(* Logix 5000 project; controller reports 1756-L63 rev 20.15; software revision 20.04; part 46 of 52 *)

        [142].log_data[50].min := 2.0290048, [142].log_data[50].max := 2.1358266, [142].log_data[50].total := 7520.501, [142].log_data[50].time := 3600.0, [142].log_data[50].minminute := 14, [142].log_data[50].maxminute := 21, [142].log_data[50].valid := 1, [142].log_data[51].time := 3600.0, [142].log_data[51].valid := 1, [142].log_data[52].min := -2.9000015, [142].log_data[52].max := 0.11999512, [142].log_data[52].total := -7928.3423, [142].log_data[52].time := 3600.0, [142].log_data[52].minminute := 8, [142].log_data[52].maxminute := 7, [142].log_data[52].valid := 1, [142].log_data[53].min := -2.4600067, [142].log_data[53].max := 0.38000488, [142].log_data[53].total := -6926.5454, [142].log_data[53].time := 3600.0, [142].log_data[53].minminute := 24, [142].log_data[53].maxminute := 13, [142].log_data[53].valid := 1, [142].log_data[54].max := 0.524, [142].log_data[54].total := 1245.6982, [142].log_data[54].time := 3600.0, [142].log_data[54].minminute := 7, [142].log_data[54].maxminute := 8, [142].log_data[54].valid := 1, [142].log_data[55].max := 0.5415, [142].log_data[55].total := 1217.0897, [142].log_data[55].time := 3600.0, [142].log_data[55].minminute := 2, [142].log_data[55].maxminute := 24, [142].log_data[55].valid := 1, [142].log_data[56].min := 0.15906787, [142].log_data[56].max := 0.15965673, [142].log_data[56].total := 573.5303, [142].log_data[56].time := 3600.0, [142].log_data[56].minminute := 45, [142].log_data[56].maxminute := 33, [142].log_data[56].valid := 1, [142].log_data[57].min := 0.19345811, [142].log_data[57].max := 0.19534253, [142].log_data[57].total := 701.22565, [142].log_data[57].time := 3600.0, [142].log_data[57].minminute := 53, [142].log_data[57].valid := 1, [142].log_data[58].time := 3600.0, [142].log_data[58].valid := 1, [142].log_data[59].time := 3600.0, [142].log_data[59].valid := 1, [142].log_data[60].valid := 1, [142].log_data[61].valid := 1, [142].log_data[62].valid := 1, [142].log_data[63].valid := 1, [142].log_data[64].valid := 1, [142].log_data[65].valid := 1, [142].log_data[66].valid := 1, [142].log_data[67].valid := 1,
        [142].log_data[68].valid := 1, [142].log_data[69].valid := 1, [142].log_data[70].valid := 1, [142].log_data[71].valid := 1, [142].log_data[72].valid := 1, [142].log_data[73].valid := 1, [142].log_data[74].valid := 1, [142].log_data[75].valid := 1, [142].log_data[76].valid := 1, [142].log_data[77].valid := 1, [142].log_data[78].valid := 1, [142].log_data[79].valid := 1, [142].log_data[80].valid := 1, [142].log_data[81].valid := 1, [142].log_data[82].valid := 1, [142].log_data[83].valid := 1, [142].log_data[84].valid := 1, [142].log_data[85].valid := 1, [142].log_data[86].valid := 1, [142].log_data[87].valid := 1, [142].log_data[88].valid := 1, [142].log_data[89].valid := 1, [142].log_data[90].valid := 1, [142].log_data[91].valid := 1, [142].log_data[92].valid := 1, [142].log_data[93].valid := 1, [142].log_data[94].valid := 1, [142].log_data[95].valid := 1, [142].log_data[96].valid := 1, [142].log_data[97].valid := 1, [142].log_data[98].valid := 1, [142].log_data[99].valid := 1, [142].log_data[100].valid := 1, [142].log_data[101].valid := 1, [142].log_data[102].valid := 1, [142].log_data[103].valid := 1, [142].log_data[104].valid := 1, [142].log_data[105].valid := 1, [142].log_data[106].valid := 1, [142].log_data[107].valid := 1, [142].log_data[108].valid := 1, [142].log_data[109].valid := 1, [142].log_data[110].valid := 1, [142].log_data[111].valid := 1, [142].log_data[112].valid := 1, [142].log_data[113].valid := 1, [142].log_data[114].valid := 1, [142].log_data[115].valid := 1, [142].log_data[116].valid := 1, [142].log_data[117].valid := 1, [142].log_data[118].valid := 1, [142].log_data[119].valid := 1, [142].log_data[120].valid := 1, [142].log_data[121].valid := 1, [142].log_data[122].valid := 1, [142].log_data[123].valid := 1, [142].log_data[124].valid := 1, [142].time.Year := 2023, [142].time.Month := 1, [142].time.Day := 19,
        [142].time.Hour := 1, [142].time.Minute := 59, [142].time.Second := 59, [143].log_data[0].min := 1.0, [143].log_data[0].max := 1.0, [143].log_data[0].total := 3600.0, [143].log_data[0].time := 3600.0, [143].log_data[0].valid := 1, [143].log_data[1].time := 3600.0, [143].log_data[1].valid := 1, [143].log_data[2].time := 3600.0, [143].log_data[2].valid := 1, [143].log_data[3].time := 3600.0, [143].log_data[3].valid := 1, [143].log_data[4].time := 3600.0, [143].log_data[4].valid := 1, [143].log_data[5].time := 3600.0, [143].log_data[5].valid := 1, [143].log_data[6].time := 3600.0, [143].log_data[6].valid := 1, [143].log_data[7].time := 3600.0, [143].log_data[7].valid := 1, [143].log_data[8].min := 1.0, [143].log_data[8].max := 1.0, [143].log_data[8].total := 3600.0, [143].log_data[8].time := 3600.0, [143].log_data[8].valid := 1, [143].log_data[9].min := 1.0, [143].log_data[9].max := 1.0, [143].log_data[9].total := 3600.0, [143].log_data[9].time := 3600.0, [143].log_data[9].valid := 1, [143].log_data[10].min := 1.0, [143].log_data[10].max := 1.0, [143].log_data[10].total := 3600.0, [143].log_data[10].time := 3600.0, [143].log_data[10].valid := 1, [143].log_data[11].time := 3600.0, [143].log_data[11].valid := 1, [143].log_data[12].min := 1.0, [143].log_data[12].max := 1.0, [143].log_data[12].total := 3600.0, [143].log_data[12].time := 3600.0, [143].log_data[12].valid := 1, [143].log_data[13].min := 1.0, [143].log_data[13].max := 1.0, [143].log_data[13].total := 3600.0, [143].log_data[13].time := 3600.0, [143].log_data[13].valid := 1, [143].log_data[14].time := 3600.0, [143].log_data[14].valid := 1, [143].log_data[15].time := 3600.0, [143].log_data[15].valid := 1, [143].log_data[16].time := 3600.0, [143].log_data[16].valid := 1, [143].log_data[17].min := 1.0, [143].log_data[17].max := 1.0, [143].log_data[17].total := 3600.0, [143].log_data[17].time := 3600.0, [143].log_data[17].valid := 1,
        [143].log_data[18].time := 3600.0, [143].log_data[18].valid := 1, [143].log_data[19].time := 3600.0, [143].log_data[19].valid := 1, [143].log_data[20].time := 3600.0, [143].log_data[20].valid := 1, [143].log_data[21].min := 1.0, [143].log_data[21].max := 1.0, [143].log_data[21].total := 3600.0, [143].log_data[21].time := 3600.0, [143].log_data[21].valid := 1, [143].log_data[22].time := 3600.0, [143].log_data[22].valid := 1, [143].log_data[23].time := 3600.0, [143].log_data[23].valid := 1, [143].log_data[24].time := 3600.0, [143].log_data[24].valid := 1, [143].log_data[25].time := 3600.0, [143].log_data[25].valid := 1, [143].log_data[26].time := 3600.0, [143].log_data[26].valid := 1, [143].log_data[27].time := 3600.0, [143].log_data[27].valid := 1, [143].log_data[28].time := 3600.0, [143].log_data[28].valid := 1, [143].log_data[29].min := 1.0, [143].log_data[29].max := 1.0, [143].log_data[29].total := 3600.0, [143].log_data[29].time := 3600.0, [143].log_data[29].valid := 1, [143].log_data[30].min := 1.0, [143].log_data[30].max := 1.0, [143].log_data[30].total := 3600.0, [143].log_data[30].time := 3600.0, [143].log_data[30].valid := 1, [143].log_data[31].max := 1.0, [143].log_data[31].total := 1464.2471, [143].log_data[31].time := 3600.0, [143].log_data[31].maxminute := 11, [143].log_data[31].valid := 1, [143].log_data[32].max := 1.0, [143].log_data[32].total := 1629.998, [143].log_data[32].time := 3600.0, [143].log_data[32].maxminute := 1, [143].log_data[32].valid := 1, [143].log_data[33].time := 3600.0, [143].log_data[33].valid := 1, [143].log_data[34].time := 3600.0, [143].log_data[34].valid := 1, [143].log_data[35].max := 1.0, [143].log_data[35].total := 1629.498, [143].log_data[35].time := 3600.0, [143].log_data[35].maxminute := 6, [143].log_data[35].valid := 1, [143].log_data[36].max := 1.0, [143].log_data[36].total := 1440.7471, [143].log_data[36].time := 3600.0, [143].log_data[36].minminute := 5, [143].log_data[36].valid := 1, [143].log_data[37].time := 3600.0,
        [143].log_data[37].valid := 1, [143].log_data[38].time := 3600.0, [143].log_data[38].valid := 1, [143].log_data[39].min := 0.9961195, [143].log_data[39].max := 1.0054238, [143].log_data[39].total := 3604.2942, [143].log_data[39].time := 3600.0, [143].log_data[39].minminute := 29, [143].log_data[39].maxminute := 50, [143].log_data[39].valid := 1, [143].log_data[40].min := 7.602789, [143].log_data[40].max := 7.622027, [143].log_data[40].total := 27405.582, [143].log_data[40].time := 3600.0, [143].log_data[40].minminute := 5, [143].log_data[40].maxminute := 10, [143].log_data[40].valid := 1, [143].log_data[41].min := 0.02273633, [143].log_data[41].max := 0.023128908, [143].log_data[41].total := 82.62436, [143].log_data[41].time := 3600.0, [143].log_data[41].valid := 1, [143].log_data[42].min := 2.291525, [143].log_data[42].max := 2.296236, [143].log_data[42].total := 8257.919, [143].log_data[42].time := 3600.0, [143].log_data[42].minminute := 2, [143].log_data[42].maxminute := 20, [143].log_data[42].valid := 1, [143].log_data[43].min := -0.27999878, [143].log_data[43].max := -0.26000214, [143].log_data[43].total := -1007.4526, [143].log_data[43].time := 3600.0, [143].log_data[43].maxminute := 8, [143].log_data[43].valid := 1, [143].log_data[44].min := -0.3199997, [143].log_data[44].max := -0.30000305, [143].log_data[44].total := -1092.692, [143].log_data[44].time := 3600.0, [143].log_data[44].valid := 1, [143].log_data[45].time := 3600.0, [143].log_data[45].valid := 1, [143].log_data[46].time := 3600.0, [143].log_data[46].valid := 1, [143].log_data[47].time := 3600.0, [143].log_data[47].valid := 1, [143].log_data[48].min := 6.7536335, [143].log_data[48].max := 6.7967777, [143].log_data[48].total := 24351.693, [143].log_data[48].time := 3600.0, [143].log_data[48].minminute := 54, [143].log_data[48].maxminute := 1, [143].log_data[48].valid := 1, [143].log_data[49].min := 8.710789, [143].log_data[49].max := 9.616479, [143].log_data[49].total := 33962.16, [143].log_data[49].time := 3600.0, [143].log_data[49].maxminute := 42, [143].log_data[49].valid := 1, [143].log_data[50].min := 2.0009744,
        [143].log_data[50].max := 2.0865965, [143].log_data[50].total := 7354.9937, [143].log_data[50].time := 3600.0, [143].log_data[50].minminute := 59, [143].log_data[50].valid := 1, [143].log_data[51].time := 3600.0, [143].log_data[51].valid := 1, [143].log_data[52].min := -2.8199997, [143].log_data[52].max := 0.11999512, [143].log_data[52].total := -7782.8364, [143].log_data[52].time := 3600.0, [143].log_data[52].minminute := 32, [143].log_data[52].maxminute := 11, [143].log_data[52].valid := 1, [143].log_data[53].min := -2.6200027, [143].log_data[53].max := 0.33999634, [143].log_data[53].total := -6983.5625, [143].log_data[53].time := 3600.0, [143].log_data[53].minminute := 48, [143].log_data[53].maxminute := 16, [143].log_data[53].valid := 1, [143].log_data[54].max := 0.5265, [143].log_data[54].total := 1226.1595, [143].log_data[54].time := 3600.0, [143].log_data[54].maxminute := 32, [143].log_data[54].valid := 1, [143].log_data[55].max := 0.55149996, [143].log_data[55].total := 1217.2601, [143].log_data[55].time := 3600.0, [143].log_data[55].minminute := 5, [143].log_data[55].maxminute := 48, [143].log_data[55].valid := 1, [143].log_data[56].min := 0.15918565, [143].log_data[56].max := 0.15961748, [143].log_data[56].total := 573.6516, [143].log_data[56].time := 3600.0, [143].log_data[56].maxminute := 29, [143].log_data[56].valid := 1, [143].log_data[57].min := 0.1933796, [143].log_data[57].max := 0.19381143, [143].log_data[57].total := 696.8782, [143].log_data[57].time := 3600.0, [143].log_data[57].minminute := 28, [143].log_data[57].maxminute := 7, [143].log_data[57].valid := 1, [143].log_data[58].time := 3600.0, [143].log_data[58].valid := 1, [143].log_data[59].time := 3600.0, [143].log_data[59].valid := 1, [143].log_data[60].valid := 1, [143].log_data[61].valid := 1, [143].log_data[62].valid := 1, [143].log_data[63].valid := 1, [143].log_data[64].valid := 1, [143].log_data[65].valid := 1, [143].log_data[66].valid := 1, [143].log_data[67].valid := 1, [143].log_data[68].valid := 1, [143].log_data[69].valid := 1, [143].log_data[70].valid := 1,
        [143].log_data[71].valid := 1, [143].log_data[72].valid := 1, [143].log_data[73].valid := 1, [143].log_data[74].valid := 1, [143].log_data[75].valid := 1, [143].log_data[76].valid := 1, [143].log_data[77].valid := 1, [143].log_data[78].valid := 1, [143].log_data[79].valid := 1, [143].log_data[80].valid := 1, [143].log_data[81].valid := 1, [143].log_data[82].valid := 1, [143].log_data[83].valid := 1, [143].log_data[84].valid := 1, [143].log_data[85].valid := 1, [143].log_data[86].valid := 1, [143].log_data[87].valid := 1, [143].log_data[88].valid := 1, [143].log_data[89].valid := 1, [143].log_data[90].valid := 1, [143].log_data[91].valid := 1, [143].log_data[92].valid := 1, [143].log_data[93].valid := 1, [143].log_data[94].valid := 1, [143].log_data[95].valid := 1, [143].log_data[96].valid := 1, [143].log_data[97].valid := 1, [143].log_data[98].valid := 1, [143].log_data[99].valid := 1, [143].log_data[100].valid := 1, [143].log_data[101].valid := 1, [143].log_data[102].valid := 1, [143].log_data[103].valid := 1, [143].log_data[104].valid := 1, [143].log_data[105].valid := 1, [143].log_data[106].valid := 1, [143].log_data[107].valid := 1, [143].log_data[108].valid := 1, [143].log_data[109].valid := 1, [143].log_data[110].valid := 1, [143].log_data[111].valid := 1, [143].log_data[112].valid := 1, [143].log_data[113].valid := 1, [143].log_data[114].valid := 1, [143].log_data[115].valid := 1, [143].log_data[116].valid := 1, [143].log_data[117].valid := 1, [143].log_data[118].valid := 1, [143].log_data[119].valid := 1, [143].log_data[120].valid := 1, [143].log_data[121].valid := 1, [143].log_data[122].valid := 1, [143].log_data[123].valid := 1, [143].log_data[124].valid := 1, [143].time.Year := 2023, [143].time.Month := 1, [143].time.Day := 19, [143].time.Hour := 2, [143].time.Minute := 59, [143].time.Second := 59,
        [144].log_data[0].min := 1.0, [144].log_data[0].max := 1.0, [144].log_data[0].total := 3600.0, [144].log_data[0].time := 3600.0, [144].log_data[0].valid := 1, [144].log_data[1].time := 3600.0, [144].log_data[1].valid := 1, [144].log_data[2].time := 3600.0, [144].log_data[2].valid := 1, [144].log_data[3].time := 3600.0, [144].log_data[3].valid := 1, [144].log_data[4].time := 3600.0, [144].log_data[4].valid := 1, [144].log_data[5].time := 3600.0, [144].log_data[5].valid := 1, [144].log_data[6].time := 3600.0, [144].log_data[6].valid := 1, [144].log_data[7].time := 3600.0, [144].log_data[7].valid := 1, [144].log_data[8].max := 1.0, [144].log_data[8].total := 22.251, [144].log_data[8].time := 3600.0, [144].log_data[8].valid := 1, [144].log_data[9].max := 1.0, [144].log_data[9].total := 22.251, [144].log_data[9].time := 3600.0, [144].log_data[9].valid := 1, [144].log_data[10].min := 1.0, [144].log_data[10].max := 1.0, [144].log_data[10].total := 3600.0, [144].log_data[10].time := 3600.0, [144].log_data[10].valid := 1, [144].log_data[11].time := 3600.0, [144].log_data[11].valid := 1, [144].log_data[12].min := 1.0, [144].log_data[12].max := 1.0, [144].log_data[12].total := 3600.0, [144].log_data[12].time := 3600.0, [144].log_data[12].valid := 1, [144].log_data[13].min := 1.0, [144].log_data[13].max := 1.0, [144].log_data[13].total := 3600.0, [144].log_data[13].time := 3600.0, [144].log_data[13].valid := 1, [144].log_data[14].time := 3600.0, [144].log_data[14].valid := 1, [144].log_data[15].time := 3600.0, [144].log_data[15].valid := 1, [144].log_data[16].time := 3600.0, [144].log_data[16].valid := 1, [144].log_data[17].min := 1.0, [144].log_data[17].max := 1.0, [144].log_data[17].total := 3600.0, [144].log_data[17].time := 3600.0, [144].log_data[17].valid := 1, [144].log_data[18].time := 3600.0, [144].log_data[18].valid := 1, [144].log_data[19].time := 3600.0, [144].log_data[19].valid := 1, [144].log_data[20].time := 3600.0,
        [144].log_data[20].valid := 1, [144].log_data[21].min := 1.0, [144].log_data[21].max := 1.0, [144].log_data[21].total := 3600.0, [144].log_data[21].time := 3600.0, [144].log_data[21].valid := 1, [144].log_data[22].time := 3600.0, [144].log_data[22].valid := 1, [144].log_data[23].time := 3600.0, [144].log_data[23].valid := 1, [144].log_data[24].time := 3600.0, [144].log_data[24].valid := 1, [144].log_data[25].time := 3600.0, [144].log_data[25].valid := 1, [144].log_data[26].time := 3600.0, [144].log_data[26].valid := 1, [144].log_data[27].time := 3600.0, [144].log_data[27].valid := 1, [144].log_data[28].time := 3600.0, [144].log_data[28].valid := 1, [144].log_data[29].min := 1.0, [144].log_data[29].max := 1.0, [144].log_data[29].total := 3600.0, [144].log_data[29].time := 3600.0, [144].log_data[29].valid := 1, [144].log_data[30].min := 1.0, [144].log_data[30].max := 1.0, [144].log_data[30].total := 3600.0, [144].log_data[30].time := 3600.0, [144].log_data[30].valid := 1, [144].log_data[31].max := 1.0, [144].log_data[31].total := 26.0, [144].log_data[31].time := 3600.0, [144].log_data[31].valid := 1, [144].log_data[32].time := 3600.0, [144].log_data[32].valid := 1, [144].log_data[33].time := 3600.0, [144].log_data[33].valid := 1, [144].log_data[34].time := 3600.0, [144].log_data[34].valid := 1, [144].log_data[35].time := 3600.0, [144].log_data[35].valid := 1, [144].log_data[36].max := 1.0, [144].log_data[36].total := 26.0, [144].log_data[36].time := 3600.0, [144].log_data[36].valid := 1, [144].log_data[37].time := 3600.0, [144].log_data[37].valid := 1, [144].log_data[38].time := 3600.0, [144].log_data[38].valid := 1, [144].log_data[39].min := 0.99623734, [144].log_data[39].max := 1.0056593, [144].log_data[39].total := 3605.3367, [144].log_data[39].time := 3600.0, [144].log_data[39].minminute := 48, [144].log_data[39].maxminute := 56, [144].log_data[39].valid := 1, [144].log_data[40].min := 7.5972934, [144].log_data[40].max := 7.6363163, [144].log_data[40].total := 27399.168,
        [144].log_data[40].time := 3600.0, [144].log_data[40].minminute := 26, [144].log_data[40].maxminute := 33, [144].log_data[40].valid := 1, [144].log_data[41].min := 0.02273633, [144].log_data[41].max := 0.023128908, [144].log_data[41].total := 82.62523, [144].log_data[41].time := 3600.0, [144].log_data[41].valid := 1, [144].log_data[42].min := 2.2910538, [144].log_data[42].max := 2.2958827, [144].log_data[42].total := 8257.894, [144].log_data[42].time := 3600.0, [144].log_data[42].minminute := 22, [144].log_data[42].maxminute := 8, [144].log_data[42].valid := 1, [144].log_data[43].min := -0.27999878, [144].log_data[43].max := -0.26000214, [144].log_data[43].total := -1007.2367, [144].log_data[43].time := 3600.0, [144].log_data[43].valid := 1, [144].log_data[44].min := -0.3199997, [144].log_data[44].max := -0.30000305, [144].log_data[44].total := -1086.3679, [144].log_data[44].time := 3600.0, [144].log_data[44].valid := 1, [144].log_data[45].time := 3600.0, [144].log_data[45].valid := 1, [144].log_data[46].time := 3600.0, [144].log_data[46].valid := 1, [144].log_data[47].time := 3600.0, [144].log_data[47].valid := 1, [144].log_data[48].min := 6.7519846, [144].log_data[48].max := 6.768473, [144].log_data[48].total := 24336.852, [144].log_data[48].time := 3600.0, [144].log_data[48].minminute := 2, [144].log_data[48].maxminute := 55, [144].log_data[48].valid := 1, [144].log_data[49].min := 9.541692, [144].log_data[49].max := 9.602148, [144].log_data[49].total := 34445.23, [144].log_data[49].time := 3600.0, [144].log_data[49].minminute := 5, [144].log_data[49].maxminute := 7, [144].log_data[49].valid := 1, [144].log_data[50].min := 1.9997966, [144].log_data[50].max := 2.110623, [144].log_data[50].total := 7565.291, [144].log_data[50].time := 3600.0, [144].log_data[50].maxminute := 56, [144].log_data[50].valid := 1, [144].log_data[51].time := 3600.0, [144].log_data[51].valid := 1, [144].log_data[52].min := -2.6399994, [144].log_data[52].max := -0.08000183, [144].log_data[52].total := -5223.154, [144].log_data[52].time := 3600.0, [144].log_data[52].valid := 1, [144].log_data[53].min := -2.4200058,
        [144].log_data[53].max := -0.16000366, [144].log_data[53].total := -4604.705, [144].log_data[53].time := 3600.0, [144].log_data[53].valid := 1, [144].log_data[54].max := 0.43400002, [144].log_data[54].total := 10.802108, [144].log_data[54].time := 3600.0, [144].log_data[54].valid := 1, [144].log_data[55].max := 0.4145, [144].log_data[55].total := 10.702488, [144].log_data[55].time := 3600.0, [144].log_data[55].valid := 1, [144].log_data[56].min := 0.15918565, [144].log_data[56].max := 0.15961748, [144].log_data[56].total := 573.69305, [144].log_data[56].time := 3600.0, [144].log_data[56].minminute := 11, [144].log_data[56].maxminute := 36, [144].log_data[56].valid := 1, [144].log_data[57].min := 0.19334033, [144].log_data[57].max := 0.19377217, [144].log_data[57].total := 696.698, [144].log_data[57].time := 3600.0, [144].log_data[57].minminute := 2, [144].log_data[57].maxminute := 16, [144].log_data[57].valid := 1, [144].log_data[58].time := 3600.0, [144].log_data[58].valid := 1, [144].log_data[59].time := 3600.0, [144].log_data[59].valid := 1, [144].log_data[60].valid := 1, [144].log_data[61].valid := 1, [144].log_data[62].valid := 1, [144].log_data[63].valid := 1, [144].log_data[64].valid := 1, [144].log_data[65].valid := 1, [144].log_data[66].valid := 1, [144].log_data[67].valid := 1, [144].log_data[68].valid := 1, [144].log_data[69].valid := 1, [144].log_data[70].valid := 1, [144].log_data[71].valid := 1, [144].log_data[72].valid := 1, [144].log_data[73].valid := 1, [144].log_data[74].valid := 1, [144].log_data[75].valid := 1, [144].log_data[76].valid := 1, [144].log_data[77].valid := 1, [144].log_data[78].valid := 1, [144].log_data[79].valid := 1, [144].log_data[80].valid := 1, [144].log_data[81].valid := 1, [144].log_data[82].valid := 1, [144].log_data[83].valid := 1, [144].log_data[84].valid := 1, [144].log_data[85].valid := 1, [144].log_data[86].valid := 1, [144].log_data[87].valid := 1, [144].log_data[88].valid := 1, [144].log_data[89].valid := 1,
        [144].log_data[90].valid := 1, [144].log_data[91].valid := 1, [144].log_data[92].valid := 1, [144].log_data[93].valid := 1, [144].log_data[94].valid := 1, [144].log_data[95].valid := 1, [144].log_data[96].valid := 1, [144].log_data[97].valid := 1, [144].log_data[98].valid := 1, [144].log_data[99].valid := 1, [144].log_data[100].valid := 1, [144].log_data[101].valid := 1, [144].log_data[102].valid := 1, [144].log_data[103].valid := 1, [144].log_data[104].valid := 1, [144].log_data[105].valid := 1, [144].log_data[106].valid := 1, [144].log_data[107].valid := 1, [144].log_data[108].valid := 1, [144].log_data[109].valid := 1, [144].log_data[110].valid := 1, [144].log_data[111].valid := 1, [144].log_data[112].valid := 1, [144].log_data[113].valid := 1, [144].log_data[114].valid := 1, [144].log_data[115].valid := 1, [144].log_data[116].valid := 1, [144].log_data[117].valid := 1, [144].log_data[118].valid := 1, [144].log_data[119].valid := 1, [144].log_data[120].valid := 1, [144].log_data[121].valid := 1, [144].log_data[122].valid := 1, [144].log_data[123].valid := 1, [144].log_data[124].valid := 1, [144].time.Year := 2023, [144].time.Month := 1, [144].time.Day := 19, [144].time.Hour := 3, [144].time.Minute := 59, [144].time.Second := 59, [145].log_data[0].min := 1.0, [145].log_data[0].max := 1.0, [145].log_data[0].total := 3600.0, [145].log_data[0].time := 3600.0, [145].log_data[0].valid := 1, [145].log_data[1].time := 3600.0, [145].log_data[1].valid := 1, [145].log_data[2].time := 3600.0, [145].log_data[2].valid := 1, [145].log_data[3].time := 3600.0, [145].log_data[3].valid := 1, [145].log_data[4].time := 3600.0, [145].log_data[4].valid := 1, [145].log_data[5].time := 3600.0, [145].log_data[5].valid := 1, [145].log_data[6].time := 3600.0, [145].log_data[6].valid := 1, [145].log_data[7].time := 3600.0, [145].log_data[7].valid := 1,
        [145].log_data[8].time := 3600.0, [145].log_data[8].valid := 1, [145].log_data[9].time := 3600.0, [145].log_data[9].valid := 1, [145].log_data[10].min := 1.0, [145].log_data[10].max := 1.0, [145].log_data[10].total := 3600.0, [145].log_data[10].time := 3600.0, [145].log_data[10].valid := 1, [145].log_data[11].time := 3600.0, [145].log_data[11].valid := 1, [145].log_data[12].min := 1.0, [145].log_data[12].max := 1.0, [145].log_data[12].total := 3600.0, [145].log_data[12].time := 3600.0, [145].log_data[12].valid := 1, [145].log_data[13].min := 1.0, [145].log_data[13].max := 1.0, [145].log_data[13].total := 3600.0, [145].log_data[13].time := 3600.0, [145].log_data[13].valid := 1, [145].log_data[14].time := 3600.0, [145].log_data[14].valid := 1, [145].log_data[15].time := 3600.0, [145].log_data[15].valid := 1, [145].log_data[16].time := 3600.0, [145].log_data[16].valid := 1, [145].log_data[17].min := 1.0, [145].log_data[17].max := 1.0, [145].log_data[17].total := 3600.0, [145].log_data[17].time := 3600.0, [145].log_data[17].valid := 1, [145].log_data[18].time := 3600.0, [145].log_data[18].valid := 1, [145].log_data[19].time := 3600.0, [145].log_data[19].valid := 1, [145].log_data[20].time := 3600.0, [145].log_data[20].valid := 1, [145].log_data[21].min := 1.0, [145].log_data[21].max := 1.0, [145].log_data[21].total := 3600.0, [145].log_data[21].time := 3600.0, [145].log_data[21].valid := 1, [145].log_data[22].time := 3600.0, [145].log_data[22].valid := 1, [145].log_data[23].time := 3600.0, [145].log_data[23].valid := 1, [145].log_data[24].time := 3600.0, [145].log_data[24].valid := 1, [145].log_data[25].time := 3600.0, [145].log_data[25].valid := 1, [145].log_data[26].time := 3600.0, [145].log_data[26].valid := 1, [145].log_data[27].time := 3600.0, [145].log_data[27].valid := 1, [145].log_data[28].time := 3600.0, [145].log_data[28].valid := 1, [145].log_data[29].min := 1.0, [145].log_data[29].max := 1.0, [145].log_data[29].total := 3600.0,
        [145].log_data[29].time := 3600.0, [145].log_data[29].valid := 1, [145].log_data[30].min := 1.0, [145].log_data[30].max := 1.0, [145].log_data[30].total := 3600.0, [145].log_data[30].time := 3600.0, [145].log_data[30].valid := 1, [145].log_data[31].time := 3600.0, [145].log_data[31].valid := 1, [145].log_data[32].time := 3600.0, [145].log_data[32].valid := 1, [145].log_data[33].time := 3600.0, [145].log_data[33].valid := 1, [145].log_data[34].time := 3600.0, [145].log_data[34].valid := 1, [145].log_data[35].time := 3600.0, [145].log_data[35].valid := 1, [145].log_data[36].time := 3600.0, [145].log_data[36].valid := 1, [145].log_data[37].time := 3600.0, [145].log_data[37].valid := 1, [145].log_data[38].time := 3600.0, [145].log_data[38].valid := 1, [145].log_data[39].min := 0.9967084, [145].log_data[39].max := 1.0062482, [145].log_data[39].total := 3605.411, [145].log_data[39].time := 3600.0, [145].log_data[39].maxminute := 1, [145].log_data[39].valid := 1, [145].log_data[40].min := 7.6030645, [145].log_data[40].max := 7.6250496, [145].log_data[40].total := 27410.46, [145].log_data[40].time := 3600.0, [145].log_data[40].minminute := 2, [145].log_data[40].maxminute := 3, [145].log_data[40].valid := 1, [145].log_data[41].min := 0.02273633, [145].log_data[41].max := 0.023128908, [145].log_data[41].total := 82.57975, [145].log_data[41].time := 3600.0, [145].log_data[41].valid := 1, [145].log_data[42].min := 2.290936, [145].log_data[42].max := 2.2957647, [145].log_data[42].total := 8257.829, [145].log_data[42].time := 3600.0, [145].log_data[42].minminute := 28, [145].log_data[42].maxminute := 32, [145].log_data[42].valid := 1, [145].log_data[43].min := -0.27999878, [145].log_data[43].max := -0.26000214, [145].log_data[43].total := -1001.4754, [145].log_data[43].time := 3600.0, [145].log_data[43].valid := 1, [145].log_data[44].min := -0.3199997, [145].log_data[44].max := -0.30000305, [145].log_data[44].total := -1080.5452, [145].log_data[44].time := 3600.0, [145].log_data[44].minminute := 6, [145].log_data[44].valid := 1, [145].log_data[45].time := 3600.0,
        [145].log_data[45].valid := 1, [145].log_data[46].time := 3600.0, [145].log_data[46].valid := 1, [145].log_data[47].time := 3600.0, [145].log_data[47].valid := 1, [145].log_data[48].min := 6.7662745, [145].log_data[48].max := 6.778366, [145].log_data[48].total := 24383.604, [145].log_data[48].time := 3600.0, [145].log_data[48].minminute := 1, [145].log_data[48].maxminute := 54, [145].log_data[48].valid := 1, [145].log_data[49].min := 9.56191, [145].log_data[49].max := 9.644745, [145].log_data[49].total := 34582.85, [145].log_data[49].time := 3600.0, [145].log_data[49].minminute := 5, [145].log_data[49].maxminute := 56, [145].log_data[49].valid := 1, [145].log_data[50].min := 2.1029673, [145].log_data[50].max := 2.1119182, [145].log_data[50].total := 7592.0264, [145].log_data[50].time := 3600.0, [145].log_data[50].minminute := 3, [145].log_data[50].maxminute := 54, [145].log_data[50].valid := 1, [145].log_data[51].time := 3600.0, [145].log_data[51].valid := 1, [145].log_data[52].min := -1.7000046, [145].log_data[52].max := -1.4800034, [145].log_data[52].total := -5676.7373, [145].log_data[52].time := 3600.0, [145].log_data[52].minminute := 52, [145].log_data[52].valid := 1, [145].log_data[53].min := -1.3800049, [145].log_data[53].max := -1.2000046, [145].log_data[53].total := -4570.1772, [145].log_data[53].time := 3600.0, [145].log_data[53].minminute := 1, [145].log_data[53].maxminute := 28, [145].log_data[53].valid := 1, [145].log_data[54].time := 3600.0, [145].log_data[54].valid := 1, [145].log_data[55].time := 3600.0, [145].log_data[55].valid := 1, [145].log_data[56].min := 0.15918565, [145].log_data[56].max := 0.15961748, [145].log_data[56].total := 573.68567, [145].log_data[56].time := 3600.0, [145].log_data[56].minminute := 26, [145].log_data[56].maxminute := 14, [145].log_data[56].valid := 1, [145].log_data[57].min := 0.1933796, [145].log_data[57].max := 0.19381143, [145].log_data[57].total := 696.7857, [145].log_data[57].time := 3600.0, [145].log_data[57].minminute := 17, [145].log_data[57].maxminute := 54, [145].log_data[57].valid := 1, [145].log_data[58].time := 3600.0,
        [145].log_data[58].valid := 1, [145].log_data[59].time := 3600.0, [145].log_data[59].valid := 1, [145].log_data[60].valid := 1, [145].log_data[61].valid := 1, [145].log_data[62].valid := 1, [145].log_data[63].valid := 1, [145].log_data[64].valid := 1, [145].log_data[65].valid := 1, [145].log_data[66].valid := 1, [145].log_data[67].valid := 1, [145].log_data[68].valid := 1, [145].log_data[69].valid := 1, [145].log_data[70].valid := 1, [145].log_data[71].valid := 1, [145].log_data[72].valid := 1, [145].log_data[73].valid := 1, [145].log_data[74].valid := 1, [145].log_data[75].valid := 1, [145].log_data[76].valid := 1, [145].log_data[77].valid := 1, [145].log_data[78].valid := 1, [145].log_data[79].valid := 1, [145].log_data[80].valid := 1, [145].log_data[81].valid := 1, [145].log_data[82].valid := 1, [145].log_data[83].valid := 1, [145].log_data[84].valid := 1, [145].log_data[85].valid := 1, [145].log_data[86].valid := 1, [145].log_data[87].valid := 1, [145].log_data[88].valid := 1, [145].log_data[89].valid := 1, [145].log_data[90].valid := 1, [145].log_data[91].valid := 1, [145].log_data[92].valid := 1, [145].log_data[93].valid := 1, [145].log_data[94].valid := 1, [145].log_data[95].valid := 1, [145].log_data[96].valid := 1, [145].log_data[97].valid := 1, [145].log_data[98].valid := 1, [145].log_data[99].valid := 1, [145].log_data[100].valid := 1, [145].log_data[101].valid := 1, [145].log_data[102].valid := 1, [145].log_data[103].valid := 1, [145].log_data[104].valid := 1, [145].log_data[105].valid := 1, [145].log_data[106].valid := 1, [145].log_data[107].valid := 1, [145].log_data[108].valid := 1, [145].log_data[109].valid := 1, [145].log_data[110].valid := 1, [145].log_data[111].valid := 1, [145].log_data[112].valid := 1, [145].log_data[113].valid := 1, [145].log_data[114].valid := 1, [145].log_data[115].valid := 1, [145].log_data[116].valid := 1,
        [145].log_data[117].valid := 1, [145].log_data[118].valid := 1, [145].log_data[119].valid := 1, [145].log_data[120].valid := 1, [145].log_data[121].valid := 1, [145].log_data[122].valid := 1, [145].log_data[123].valid := 1, [145].log_data[124].valid := 1, [145].time.Year := 2023, [145].time.Month := 1, [145].time.Day := 19, [145].time.Hour := 4, [145].time.Minute := 59, [145].time.Second := 59, [146].log_data[0].min := 1.0, [146].log_data[0].max := 1.0, [146].log_data[0].total := 3600.0, [146].log_data[0].time := 3600.0, [146].log_data[0].valid := 1, [146].log_data[1].max := 1.0, [146].log_data[1].total := 527.5, [146].log_data[1].time := 3600.0, [146].log_data[1].maxminute := 34, [146].log_data[1].valid := 1, [146].log_data[2].max := 1.0, [146].log_data[2].total := 524.0, [146].log_data[2].time := 3600.0, [146].log_data[2].maxminute := 34, [146].log_data[2].valid := 1, [146].log_data[3].time := 3600.0, [146].log_data[3].valid := 1, [146].log_data[4].time := 3600.0, [146].log_data[4].valid := 1, [146].log_data[5].max := 1.0, [146].log_data[5].total := 219.0, [146].log_data[5].time := 3600.0, [146].log_data[5].maxminute := 37, [146].log_data[5].valid := 1, [146].log_data[6].time := 3600.0, [146].log_data[6].valid := 1, [146].log_data[7].time := 3600.0, [146].log_data[7].valid := 1, [146].log_data[8].max := 1.0, [146].log_data[8].total := 196.0, [146].log_data[8].time := 3600.0, [146].log_data[8].maxminute := 38, [146].log_data[8].valid := 1, [146].log_data[9].max := 1.0, [146].log_data[9].total := 192.5, [146].log_data[9].time := 3600.0, [146].log_data[9].maxminute := 39, [146].log_data[9].valid := 1, [146].log_data[10].min := 1.0, [146].log_data[10].max := 1.0, [146].log_data[10].total := 3600.0, [146].log_data[10].time := 3600.0, [146].log_data[10].valid := 1, [146].log_data[11].time := 3600.0, [146].log_data[11].valid := 1, [146].log_data[12].min := 1.0,
        [146].log_data[12].max := 1.0, [146].log_data[12].total := 3600.0, [146].log_data[12].time := 3600.0, [146].log_data[12].valid := 1, [146].log_data[13].min := 1.0, [146].log_data[13].max := 1.0, [146].log_data[13].total := 3600.0, [146].log_data[13].time := 3600.0, [146].log_data[13].valid := 1, [146].log_data[14].time := 3600.0, [146].log_data[14].valid := 1, [146].log_data[15].time := 3600.0, [146].log_data[15].valid := 1, [146].log_data[16].time := 3600.0, [146].log_data[16].valid := 1, [146].log_data[17].min := 1.0, [146].log_data[17].max := 1.0, [146].log_data[17].total := 3600.0, [146].log_data[17].time := 3600.0, [146].log_data[17].valid := 1, [146].log_data[18].time := 3600.0, [146].log_data[18].valid := 1, [146].log_data[19].time := 3600.0, [146].log_data[19].valid := 1, [146].log_data[20].time := 3600.0, [146].log_data[20].valid := 1, [146].log_data[21].min := 1.0, [146].log_data[21].max := 1.0, [146].log_data[21].total := 3600.0, [146].log_data[21].time := 3600.0, [146].log_data[21].valid := 1, [146].log_data[22].time := 3600.0, [146].log_data[22].valid := 1, [146].log_data[23].time := 3600.0, [146].log_data[23].valid := 1, [146].log_data[24].time := 3600.0, [146].log_data[24].valid := 1, [146].log_data[25].time := 3600.0, [146].log_data[25].valid := 1, [146].log_data[26].time := 3600.0, [146].log_data[26].valid := 1, [146].log_data[27].time := 3600.0, [146].log_data[27].valid := 1, [146].log_data[28].time := 3600.0, [146].log_data[28].valid := 1, [146].log_data[29].min := 1.0, [146].log_data[29].max := 1.0, [146].log_data[29].total := 3600.0, [146].log_data[29].time := 3600.0, [146].log_data[29].valid := 1, [146].log_data[30].min := 1.0, [146].log_data[30].max := 1.0, [146].log_data[30].total := 3600.0, [146].log_data[30].time := 3600.0, [146].log_data[30].valid := 1, [146].log_data[31].max := 1.0, [146].log_data[31].total := 16.749, [146].log_data[31].time := 3600.0, [146].log_data[31].maxminute := 39, [146].log_data[31].valid := 1,
        [146].log_data[32].max := 1.0, [146].log_data[32].total := 127.998, [146].log_data[32].time := 3600.0, [146].log_data[32].maxminute := 39, [146].log_data[32].valid := 1, [146].log_data[33].max := 1.0, [146].log_data[33].total := 851.0, [146].log_data[33].time := 3600.0, [146].log_data[33].maxminute := 22, [146].log_data[33].valid := 1, [146].log_data[34].max := 1.0, [146].log_data[34].total := 977.749, [146].log_data[34].time := 3600.0, [146].log_data[34].maxminute := 22, [146].log_data[34].valid := 1, [146].log_data[35].max := 1.0, [146].log_data[35].total := 132.249, [146].log_data[35].time := 3600.0, [146].log_data[35].maxminute := 40, [146].log_data[35].valid := 1, [146].log_data[36].time := 3600.0, [146].log_data[36].valid := 1, [146].log_data[37].max := 7.264285, [146].log_data[37].total := 3291.6736, [146].log_data[37].time := 3600.0, [146].log_data[37].maxminute := 36, [146].log_data[37].valid := 1, [146].log_data[38].time := 3600.0, [146].log_data[38].valid := 1, [146].log_data[39].min := 0.9957663, [146].log_data[39].max := 1.02203, [146].log_data[39].total := 3609.575, [146].log_data[39].time := 3600.0, [146].log_data[39].minminute := 54, [146].log_data[39].maxminute := 37, [146].log_data[39].valid := 1, [146].log_data[40].min := 7.607462, [146].log_data[40].max := 7.617629, [146].log_data[40].total := 27412.824, [146].log_data[40].time := 3600.0, [146].log_data[40].minminute := 22, [146].log_data[40].maxminute := 25, [146].log_data[40].valid := 1, [146].log_data[41].min := 0.022540038, [146].log_data[41].max := 0.023128908, [146].log_data[41].total := 82.52068, [146].log_data[41].time := 3600.0, [146].log_data[41].minminute := 24, [146].log_data[41].valid := 1, [146].log_data[42].min := 2.2910538, [146].log_data[42].max := 2.296236, [146].log_data[42].total := 8257.656, [146].log_data[42].time := 3600.0, [146].log_data[42].minminute := 3, [146].log_data[42].maxminute := 7, [146].log_data[42].valid := 1, [146].log_data[43].min := -0.27999878, [146].log_data[43].max := -0.26000214, [146].log_data[43].total := -955.7776, [146].log_data[43].time := 3600.0,
        [146].log_data[43].valid := 1, [146].log_data[44].min := -0.30000305, [146].log_data[44].max := -0.27999878, [146].log_data[44].total := -1080.086, [146].log_data[44].time := 3600.0, [146].log_data[44].maxminute := 44, [146].log_data[44].valid := 1, [146].log_data[45].time := 3600.0, [146].log_data[45].valid := 1, [146].log_data[46].time := 3600.0, [146].log_data[46].valid := 1, [146].log_data[47].time := 3600.0, [146].log_data[47].valid := 1, [146].log_data[48].min := 6.666519, [146].log_data[48].max := 6.9240146, [146].log_data[48].total := 24420.646, [146].log_data[48].time := 3600.0, [146].log_data[48].minminute := 59, [146].log_data[48].maxminute := 39, [146].log_data[48].valid := 1, [146].log_data[49].min := 6.6440372, [146].log_data[49].max := 9.671244, [146].log_data[49].total := 32584.168, [146].log_data[49].time := 3600.0, [146].log_data[49].minminute := 59, [146].log_data[49].maxminute := 28, [146].log_data[49].valid := 1, [146].log_data[50].min := 1.99591, [146].log_data[50].max := 2.150784, [146].log_data[50].total := 7577.36, [146].log_data[50].time := 3600.0, [146].log_data[50].minminute := 42, [146].log_data[50].maxminute := 38, [146].log_data[50].valid := 1, [146].log_data[51].max := 3.0289998, [146].log_data[51].total := 2932.7834, [146].log_data[51].time := 3600.0, [146].log_data[51].maxminute := 23, [146].log_data[51].valid := 1, [146].log_data[52].min := -6.0199966, [146].log_data[52].max := -0.30000305, [146].log_data[52].total := -6353.1074, [146].log_data[52].time := 3600.0, [146].log_data[52].minminute := 39, [146].log_data[52].maxminute := 42, [146].log_data[52].valid := 1, [146].log_data[53].min := -5.0, [146].log_data[53].max := -0.16000366, [146].log_data[53].total := -5862.117, [146].log_data[53].time := 3600.0, [146].log_data[53].minminute := 40, [146].log_data[53].maxminute := 42, [146].log_data[53].valid := 1, [146].log_data[54].max := 0.539, [146].log_data[54].total := 52.01471, [146].log_data[54].time := 3600.0, [146].log_data[54].maxminute := 39, [146].log_data[54].valid := 1, [146].log_data[55].max := 0.52, [146].log_data[55].total := 51.096313,
        [146].log_data[55].time := 3600.0, [146].log_data[55].maxminute := 40, [146].log_data[55].valid := 1, [146].log_data[56].min := 0.15914638, [146].log_data[56].max := 0.15961748, [146].log_data[56].total := 573.68787, [146].log_data[56].time := 3600.0, [146].log_data[56].minminute := 12, [146].log_data[56].maxminute := 20, [146].log_data[56].valid := 1, [146].log_data[57].min := 0.1933796, [146].log_data[57].max := 0.19381143, [146].log_data[57].total := 696.8931, [146].log_data[57].time := 3600.0, [146].log_data[57].minminute := 2, [146].log_data[57].maxminute := 6, [146].log_data[57].valid := 1, [146].log_data[58].time := 3600.0, [146].log_data[58].valid := 1, [146].log_data[59].time := 3600.0, [146].log_data[59].valid := 1, [146].log_data[60].valid := 1, [146].log_data[61].valid := 1, [146].log_data[62].valid := 1, [146].log_data[63].valid := 1, [146].log_data[64].valid := 1, [146].log_data[65].valid := 1, [146].log_data[66].valid := 1, [146].log_data[67].valid := 1, [146].log_data[68].valid := 1, [146].log_data[69].valid := 1, [146].log_data[70].valid := 1, [146].log_data[71].valid := 1, [146].log_data[72].valid := 1, [146].log_data[73].valid := 1, [146].log_data[74].valid := 1, [146].log_data[75].valid := 1, [146].log_data[76].valid := 1, [146].log_data[77].valid := 1, [146].log_data[78].valid := 1, [146].log_data[79].valid := 1, [146].log_data[80].valid := 1, [146].log_data[81].valid := 1, [146].log_data[82].valid := 1, [146].log_data[83].valid := 1, [146].log_data[84].valid := 1, [146].log_data[85].valid := 1, [146].log_data[86].valid := 1, [146].log_data[87].valid := 1, [146].log_data[88].valid := 1, [146].log_data[89].valid := 1, [146].log_data[90].valid := 1, [146].log_data[91].valid := 1, [146].log_data[92].valid := 1, [146].log_data[93].valid := 1, [146].log_data[94].valid := 1, [146].log_data[95].valid := 1, [146].log_data[96].valid := 1, [146].log_data[97].valid := 1, [146].log_data[98].valid := 1,
        [146].log_data[99].valid := 1, [146].log_data[100].valid := 1, [146].log_data[101].valid := 1, [146].log_data[102].valid := 1, [146].log_data[103].valid := 1, [146].log_data[104].valid := 1, [146].log_data[105].valid := 1, [146].log_data[106].valid := 1, [146].log_data[107].valid := 1, [146].log_data[108].valid := 1, [146].log_data[109].valid := 1, [146].log_data[110].valid := 1, [146].log_data[111].valid := 1, [146].log_data[112].valid := 1, [146].log_data[113].valid := 1, [146].log_data[114].valid := 1, [146].log_data[115].valid := 1, [146].log_data[116].valid := 1, [146].log_data[117].valid := 1, [146].log_data[118].valid := 1, [146].log_data[119].valid := 1, [146].log_data[120].valid := 1, [146].log_data[121].valid := 1, [146].log_data[122].valid := 1, [146].log_data[123].valid := 1, [146].log_data[124].valid := 1, [146].time.Year := 2023, [146].time.Month := 1, [146].time.Day := 19, [146].time.Hour := 5, [146].time.Minute := 59, [146].time.Second := 59, [147].log_data[0].min := 1.0, [147].log_data[0].max := 1.0, [147].log_data[0].total := 3600.0, [147].log_data[0].time := 3600.0, [147].log_data[0].valid := 1, [147].log_data[1].time := 3600.0, [147].log_data[1].valid := 1, [147].log_data[2].time := 3600.0, [147].log_data[2].valid := 1, [147].log_data[3].time := 3600.0, [147].log_data[3].valid := 1, [147].log_data[4].time := 3600.0, [147].log_data[4].valid := 1, [147].log_data[5].time := 3600.0, [147].log_data[5].valid := 1, [147].log_data[6].time := 3600.0, [147].log_data[6].valid := 1, [147].log_data[7].time := 3600.0, [147].log_data[7].valid := 1, [147].log_data[8].time := 3600.0, [147].log_data[8].valid := 1, [147].log_data[9].time := 3600.0, [147].log_data[9].valid := 1, [147].log_data[10].min := 1.0, [147].log_data[10].max := 1.0, [147].log_data[10].total := 3600.0, [147].log_data[10].time := 3600.0, [147].log_data[10].valid := 1,
        [147].log_data[11].time := 3600.0, [147].log_data[11].valid := 1, [147].log_data[12].min := 1.0, [147].log_data[12].max := 1.0, [147].log_data[12].total := 3600.0, [147].log_data[12].time := 3600.0, [147].log_data[12].valid := 1, [147].log_data[13].min := 1.0, [147].log_data[13].max := 1.0, [147].log_data[13].total := 3600.0, [147].log_data[13].time := 3600.0, [147].log_data[13].valid := 1, [147].log_data[14].time := 3600.0, [147].log_data[14].valid := 1, [147].log_data[15].time := 3600.0, [147].log_data[15].valid := 1, [147].log_data[16].time := 3600.0, [147].log_data[16].valid := 1, [147].log_data[17].min := 1.0, [147].log_data[17].max := 1.0, [147].log_data[17].total := 3600.0, [147].log_data[17].time := 3600.0, [147].log_data[17].valid := 1, [147].log_data[18].time := 3600.0, [147].log_data[18].valid := 1, [147].log_data[19].time := 3600.0, [147].log_data[19].valid := 1, [147].log_data[20].time := 3600.0, [147].log_data[20].valid := 1, [147].log_data[21].min := 1.0, [147].log_data[21].max := 1.0, [147].log_data[21].total := 3600.0, [147].log_data[21].time := 3600.0, [147].log_data[21].valid := 1, [147].log_data[22].time := 3600.0, [147].log_data[22].valid := 1, [147].log_data[23].time := 3600.0, [147].log_data[23].valid := 1, [147].log_data[24].time := 3600.0, [147].log_data[24].valid := 1, [147].log_data[25].time := 3600.0, [147].log_data[25].valid := 1, [147].log_data[26].time := 3600.0, [147].log_data[26].valid := 1, [147].log_data[27].time := 3600.0, [147].log_data[27].valid := 1, [147].log_data[28].time := 3600.0, [147].log_data[28].valid := 1, [147].log_data[29].min := 1.0, [147].log_data[29].max := 1.0, [147].log_data[29].total := 3600.0, [147].log_data[29].time := 3600.0, [147].log_data[29].valid := 1, [147].log_data[30].min := 1.0, [147].log_data[30].max := 1.0, [147].log_data[30].total := 3600.0, [147].log_data[30].time := 3600.0, [147].log_data[30].valid := 1, [147].log_data[31].time := 3600.0, [147].log_data[31].valid := 1,
        [147].log_data[32].time := 3600.0, [147].log_data[32].valid := 1, [147].log_data[33].time := 3600.0, [147].log_data[33].valid := 1, [147].log_data[34].time := 3600.0, [147].log_data[34].valid := 1, [147].log_data[35].time := 3600.0, [147].log_data[35].valid := 1, [147].log_data[36].time := 3600.0, [147].log_data[36].valid := 1, [147].log_data[37].time := 3600.0, [147].log_data[37].valid := 1, [147].log_data[38].time := 3600.0, [147].log_data[38].valid := 1, [147].log_data[39].min := 0.9956484, [147].log_data[39].max := 1.0051882, [147].log_data[39].total := 3602.7424, [147].log_data[39].time := 3600.0, [147].log_data[39].minminute := 25, [147].log_data[39].maxminute := 58, [147].log_data[39].valid := 1, [147].log_data[40].min := 7.6099358, [147].log_data[40].max := 7.6148815, [147].log_data[40].total := 27409.361, [147].log_data[40].time := 3600.0, [147].log_data[40].minminute := 31, [147].log_data[40].maxminute := 3, [147].log_data[40].valid := 1, [147].log_data[41].min := 0.022540038, [147].log_data[41].max := 0.023128908, [147].log_data[41].total := 82.322296, [147].log_data[41].time := 3600.0, [147].log_data[41].minminute := 5, [147].log_data[41].valid := 1, [147].log_data[42].min := 2.291407, [147].log_data[42].max := 2.2958827, [147].log_data[42].total := 8257.53, [147].log_data[42].time := 3600.0, [147].log_data[42].minminute := 12, [147].log_data[42].maxminute := 7, [147].log_data[42].valid := 1, [147].log_data[43].min := -0.27999878, [147].log_data[43].max := -0.26000214, [147].log_data[43].total := -936.6149, [147].log_data[43].time := 3600.0, [147].log_data[43].valid := 1, [147].log_data[44].min := -0.30000305, [147].log_data[44].max := -0.27999878, [147].log_data[44].total := -1079.0758, [147].log_data[44].time := 3600.0, [147].log_data[44].maxminute := 2, [147].log_data[44].valid := 1, [147].log_data[45].time := 3600.0, [147].log_data[45].valid := 1, [147].log_data[46].time := 3600.0, [147].log_data[46].valid := 1, [147].log_data[47].time := 3600.0, [147].log_data[47].valid := 1, [147].log_data[48].min := 6.552199, [147].log_data[48].max := 6.666794,
        [147].log_data[48].total := 23742.52, [147].log_data[48].time := 3600.0, [147].log_data[48].minminute := 16, [147].log_data[48].valid := 1, [147].log_data[49].min := 6.1886415, [147].log_data[49].max := 9.473578, [147].log_data[49].total := 28327.7, [147].log_data[49].time := 3600.0, [147].log_data[49].minminute := 12, [147].log_data[49].maxminute := 59, [147].log_data[49].valid := 1, [147].log_data[50].min := 2.1072073, [147].log_data[50].max := 2.1213403, [147].log_data[50].total := 7619.476, [147].log_data[50].time := 3600.0, [147].log_data[50].maxminute := 49, [147].log_data[50].valid := 1, [147].log_data[51].time := 3600.0, [147].log_data[51].valid := 1, [147].log_data[52].min := -1.5800018, [147].log_data[52].max := -1.4000015, [147].log_data[52].total := -5416.315, [147].log_data[52].time := 3600.0, [147].log_data[52].minminute := 11, [147].log_data[52].valid := 1, [147].log_data[53].min := -1.5200043, [147].log_data[53].max := -1.340004, [147].log_data[53].total := -5208.1646, [147].log_data[53].time := 3600.0, [147].log_data[53].minminute := 18, [147].log_data[53].valid := 1, [147].log_data[54].time := 3600.0, [147].log_data[54].valid := 1, [147].log_data[55].time := 3600.0, [147].log_data[55].valid := 1, [147].log_data[56].min := 0.15914638, [147].log_data[56].max := 0.15957822, [147].log_data[56].total := 573.5847, [147].log_data[56].time := 3600.0, [147].log_data[56].minminute := 43, [147].log_data[56].maxminute := 31, [147].log_data[56].valid := 1, [147].log_data[57].min := 0.19341885, [147].log_data[57].max := 0.19385068, [147].log_data[57].total := 696.9681, [147].log_data[57].time := 3600.0, [147].log_data[57].minminute := 35, [147].log_data[57].maxminute := 31, [147].log_data[57].valid := 1, [147].log_data[58].time := 3600.0, [147].log_data[58].valid := 1, [147].log_data[59].time := 3600.0, [147].log_data[59].valid := 1, [147].log_data[60].valid := 1, [147].log_data[61].valid := 1, [147].log_data[62].valid := 1, [147].log_data[63].valid := 1, [147].log_data[64].valid := 1, [147].log_data[65].valid := 1, [147].log_data[66].valid := 1,
        [147].log_data[67].valid := 1, [147].log_data[68].valid := 1, [147].log_data[69].valid := 1, [147].log_data[70].valid := 1, [147].log_data[71].valid := 1, [147].log_data[72].valid := 1, [147].log_data[73].valid := 1, [147].log_data[74].valid := 1, [147].log_data[75].valid := 1, [147].log_data[76].valid := 1, [147].log_data[77].valid := 1, [147].log_data[78].valid := 1, [147].log_data[79].valid := 1, [147].log_data[80].valid := 1, [147].log_data[81].valid := 1, [147].log_data[82].valid := 1, [147].log_data[83].valid := 1, [147].log_data[84].valid := 1, [147].log_data[85].valid := 1, [147].log_data[86].valid := 1, [147].log_data[87].valid := 1, [147].log_data[88].valid := 1, [147].log_data[89].valid := 1, [147].log_data[90].valid := 1, [147].log_data[91].valid := 1, [147].log_data[92].valid := 1, [147].log_data[93].valid := 1, [147].log_data[94].valid := 1, [147].log_data[95].valid := 1, [147].log_data[96].valid := 1, [147].log_data[97].valid := 1, [147].log_data[98].valid := 1, [147].log_data[99].valid := 1, [147].log_data[100].valid := 1, [147].log_data[101].valid := 1, [147].log_data[102].valid := 1, [147].log_data[103].valid := 1, [147].log_data[104].valid := 1, [147].log_data[105].valid := 1, [147].log_data[106].valid := 1, [147].log_data[107].valid := 1, [147].log_data[108].valid := 1, [147].log_data[109].valid := 1, [147].log_data[110].valid := 1, [147].log_data[111].valid := 1, [147].log_data[112].valid := 1, [147].log_data[113].valid := 1, [147].log_data[114].valid := 1, [147].log_data[115].valid := 1, [147].log_data[116].valid := 1, [147].log_data[117].valid := 1, [147].log_data[118].valid := 1, [147].log_data[119].valid := 1, [147].log_data[120].valid := 1, [147].log_data[121].valid := 1, [147].log_data[122].valid := 1, [147].log_data[123].valid := 1, [147].log_data[124].valid := 1, [147].time.Year := 2023, [147].time.Month := 1,
        [147].time.Day := 19, [147].time.Hour := 6, [147].time.Minute := 59, [147].time.Second := 59, [148].log_data[0].min := 1.0, [148].log_data[0].max := 1.0, [148].log_data[0].total := 3600.0, [148].log_data[0].time := 3600.0, [148].log_data[0].valid := 1, [148].log_data[1].time := 3600.0, [148].log_data[1].valid := 1, [148].log_data[2].time := 3600.0, [148].log_data[2].valid := 1, [148].log_data[3].time := 3600.0, [148].log_data[3].valid := 1, [148].log_data[4].time := 3600.0, [148].log_data[4].valid := 1, [148].log_data[5].time := 3600.0, [148].log_data[5].valid := 1, [148].log_data[6].time := 3600.0, [148].log_data[6].valid := 1, [148].log_data[7].time := 3600.0, [148].log_data[7].valid := 1, [148].log_data[8].time := 3600.0, [148].log_data[8].valid := 1, [148].log_data[9].time := 3600.0, [148].log_data[9].valid := 1, [148].log_data[10].min := 1.0, [148].log_data[10].max := 1.0, [148].log_data[10].total := 3600.0, [148].log_data[10].time := 3600.0, [148].log_data[10].valid := 1, [148].log_data[11].time := 3600.0, [148].log_data[11].valid := 1, [148].log_data[12].min := 1.0, [148].log_data[12].max := 1.0, [148].log_data[12].total := 3600.0, [148].log_data[12].time := 3600.0, [148].log_data[12].valid := 1, [148].log_data[13].min := 1.0, [148].log_data[13].max := 1.0, [148].log_data[13].total := 3600.0, [148].log_data[13].time := 3600.0, [148].log_data[13].valid := 1, [148].log_data[14].time := 3600.0, [148].log_data[14].valid := 1, [148].log_data[15].time := 3600.0, [148].log_data[15].valid := 1, [148].log_data[16].time := 3600.0, [148].log_data[16].valid := 1, [148].log_data[17].min := 1.0, [148].log_data[17].max := 1.0, [148].log_data[17].total := 3600.0, [148].log_data[17].time := 3600.0, [148].log_data[17].valid := 1, [148].log_data[18].time := 3600.0, [148].log_data[18].valid := 1, [148].log_data[19].time := 3600.0, [148].log_data[19].valid := 1, [148].log_data[20].time := 3600.0,
        [148].log_data[20].valid := 1, [148].log_data[21].min := 1.0, [148].log_data[21].max := 1.0, [148].log_data[21].total := 3600.0, [148].log_data[21].time := 3600.0, [148].log_data[21].valid := 1, [148].log_data[22].time := 3600.0, [148].log_data[22].valid := 1, [148].log_data[23].time := 3600.0, [148].log_data[23].valid := 1, [148].log_data[24].time := 3600.0, [148].log_data[24].valid := 1, [148].log_data[25].time := 3600.0, [148].log_data[25].valid := 1, [148].log_data[26].time := 3600.0, [148].log_data[26].valid := 1, [148].log_data[27].time := 3600.0, [148].log_data[27].valid := 1, [148].log_data[28].time := 3600.0, [148].log_data[28].valid := 1, [148].log_data[29].min := 1.0, [148].log_data[29].max := 1.0, [148].log_data[29].total := 3600.0, [148].log_data[29].time := 3600.0, [148].log_data[29].valid := 1, [148].log_data[30].min := 1.0, [148].log_data[30].max := 1.0, [148].log_data[30].total := 3600.0, [148].log_data[30].time := 3600.0, [148].log_data[30].valid := 1, [148].log_data[31].time := 3600.0, [148].log_data[31].valid := 1, [148].log_data[32].time := 3600.0, [148].log_data[32].valid := 1, [148].log_data[33].time := 3600.0, [148].log_data[33].valid := 1, [148].log_data[34].time := 3600.0, [148].log_data[34].valid := 1, [148].log_data[35].time := 3600.0, [148].log_data[35].valid := 1, [148].log_data[36].time := 3600.0, [148].log_data[36].valid := 1, [148].log_data[37].time := 3600.0, [148].log_data[37].valid := 1, [148].log_data[38].time := 3600.0, [148].log_data[38].valid := 1, [148].log_data[39].min := 0.9957663, [148].log_data[39].max := 1.0050704, [148].log_data[39].total := 3603.2383, [148].log_data[39].time := 3600.0, [148].log_data[39].minminute := 42, [148].log_data[39].maxminute := 51, [148].log_data[39].valid := 1, [148].log_data[40].min := 7.607187, [148].log_data[40].max := 7.6179047, [148].log_data[40].total := 27410.693, [148].log_data[40].time := 3600.0, [148].log_data[40].minminute := 19, [148].log_data[40].maxminute := 38, [148].log_data[40].valid := 1,
        [148].log_data[41].min := 0.022540038, [148].log_data[41].max := 0.023128908, [148].log_data[41].total := 82.39118, [148].log_data[41].time := 3600.0, [148].log_data[41].minminute := 54, [148].log_data[41].valid := 1, [148].log_data[42].min := 2.290936, [148].log_data[42].max := 2.2957647, [148].log_data[42].total := 8257.699, [148].log_data[42].time := 3600.0, [148].log_data[42].minminute := 23, [148].log_data[42].maxminute := 1, [148].log_data[42].valid := 1, [148].log_data[43].min := -0.27999878, [148].log_data[43].max := -0.26000214, [148].log_data[43].total := -935.9782, [148].log_data[43].time := 3600.0, [148].log_data[43].minminute := 7, [148].log_data[43].valid := 1, [148].log_data[44].min := -0.30000305, [148].log_data[44].max := -0.27999878, [148].log_data[44].total := -1071.6344, [148].log_data[44].time := 3600.0, [148].log_data[44].valid := 1, [148].log_data[45].time := 3600.0, [148].log_data[45].valid := 1, [148].log_data[46].time := 3600.0, [148].log_data[46].valid := 1, [148].log_data[47].time := 3600.0, [148].log_data[47].valid := 1, [148].log_data[48].min := 6.625023, [148].log_data[48].max := 6.6786103, [148].log_data[48].total := 23958.037, [148].log_data[48].time := 3600.0, [148].log_data[48].maxminute := 58, [148].log_data[48].valid := 1, [148].log_data[49].min := 9.471223, [148].log_data[49].max := 9.740337, [148].log_data[49].total := 34759.453, [148].log_data[49].time := 3600.0, [148].log_data[49].maxminute := 59, [148].log_data[49].valid := 1, [148].log_data[50].min := 2.1128604, [148].log_data[50].max := 2.122047, [148].log_data[50].total := 7628.1763, [148].log_data[50].time := 3600.0, [148].log_data[50].minminute := 13, [148].log_data[50].maxminute := 46, [148].log_data[50].valid := 1, [148].log_data[51].time := 3600.0, [148].log_data[51].valid := 1, [148].log_data[52].min := -1.5999985, [148].log_data[52].max := -1.4400024, [148].log_data[52].total := -5538.6216, [148].log_data[52].time := 3600.0, [148].log_data[52].minminute := 4, [148].log_data[52].maxminute := 1, [148].log_data[52].valid := 1, [148].log_data[53].min := -1.5200043, [148].log_data[53].max := -1.3800049,
        [148].log_data[53].total := -5204.9385, [148].log_data[53].time := 3600.0, [148].log_data[53].minminute := 3, [148].log_data[53].maxminute := 6, [148].log_data[53].valid := 1, [148].log_data[54].time := 3600.0, [148].log_data[54].valid := 1, [148].log_data[55].time := 3600.0, [148].log_data[55].valid := 1, [148].log_data[56].min := 0.15914638, [148].log_data[56].max := 0.15953897, [148].log_data[56].total := 573.5144, [148].log_data[56].time := 3600.0, [148].log_data[56].minminute := 6, [148].log_data[56].maxminute := 12, [148].log_data[56].valid := 1, [148].log_data[57].min := 0.19345811, [148].log_data[57].max := 0.19385068, [148].log_data[57].total := 697.0067, [148].log_data[57].time := 3600.0, [148].log_data[57].minminute := 4, [148].log_data[57].valid := 1, [148].log_data[58].time := 3600.0, [148].log_data[58].valid := 1, [148].log_data[59].time := 3600.0, [148].log_data[59].valid := 1, [148].log_data[60].valid := 1, [148].log_data[61].valid := 1, [148].log_data[62].valid := 1, [148].log_data[63].valid := 1, [148].log_data[64].valid := 1, [148].log_data[65].valid := 1, [148].log_data[66].valid := 1, [148].log_data[67].valid := 1, [148].log_data[68].valid := 1, [148].log_data[69].valid := 1, [148].log_data[70].valid := 1, [148].log_data[71].valid := 1, [148].log_data[72].valid := 1, [148].log_data[73].valid := 1, [148].log_data[74].valid := 1, [148].log_data[75].valid := 1, [148].log_data[76].valid := 1, [148].log_data[77].valid := 1, [148].log_data[78].valid := 1, [148].log_data[79].valid := 1, [148].log_data[80].valid := 1, [148].log_data[81].valid := 1, [148].log_data[82].valid := 1, [148].log_data[83].valid := 1, [148].log_data[84].valid := 1, [148].log_data[85].valid := 1, [148].log_data[86].valid := 1, [148].log_data[87].valid := 1, [148].log_data[88].valid := 1, [148].log_data[89].valid := 1, [148].log_data[90].valid := 1, [148].log_data[91].valid := 1, [148].log_data[92].valid := 1, [148].log_data[93].valid := 1,
        [148].log_data[94].valid := 1, [148].log_data[95].valid := 1, [148].log_data[96].valid := 1, [148].log_data[97].valid := 1, [148].log_data[98].valid := 1, [148].log_data[99].valid := 1, [148].log_data[100].valid := 1, [148].log_data[101].valid := 1, [148].log_data[102].valid := 1, [148].log_data[103].valid := 1, [148].log_data[104].valid := 1, [148].log_data[105].valid := 1, [148].log_data[106].valid := 1, [148].log_data[107].valid := 1, [148].log_data[108].valid := 1, [148].log_data[109].valid := 1, [148].log_data[110].valid := 1, [148].log_data[111].valid := 1, [148].log_data[112].valid := 1, [148].log_data[113].valid := 1, [148].log_data[114].valid := 1, [148].log_data[115].valid := 1, [148].log_data[116].valid := 1, [148].log_data[117].valid := 1, [148].log_data[118].valid := 1, [148].log_data[119].valid := 1, [148].log_data[120].valid := 1, [148].log_data[121].valid := 1, [148].log_data[122].valid := 1, [148].log_data[123].valid := 1, [148].log_data[124].valid := 1, [148].time.Year := 2023, [148].time.Month := 1, [148].time.Day := 19, [148].time.Hour := 7, [148].time.Minute := 59, [148].time.Second := 59, [149].log_data[0].min := 1.0, [149].log_data[0].max := 1.0, [149].log_data[0].total := 3599.5, [149].log_data[0].time := 3599.5, [149].log_data[0].valid := 1, [149].log_data[1].max := 1.0, [149].log_data[1].total := 570.0, [149].log_data[1].time := 3599.5, [149].log_data[1].maxminute := 47, [149].log_data[1].valid := 1, [149].log_data[2].max := 1.0, [149].log_data[2].total := 566.5, [149].log_data[2].time := 3599.5, [149].log_data[2].maxminute := 47, [149].log_data[2].valid := 1, [149].log_data[3].time := 3599.5, [149].log_data[3].valid := 1, [149].log_data[4].time := 3599.5, [149].log_data[4].valid := 1, [149].log_data[5].max := 1.0, [149].log_data[5].total := 247.0, [149].log_data[5].time := 3599.5, [149].log_data[5].maxminute := 50,
        [149].log_data[5].valid := 1, [149].log_data[6].time := 3599.5, [149].log_data[6].valid := 1, [149].log_data[7].time := 3599.5, [149].log_data[7].valid := 1, [149].log_data[8].max := 1.0, [149].log_data[8].total := 527.249, [149].log_data[8].time := 3599.5, [149].log_data[8].maxminute := 51, [149].log_data[8].valid := 1, [149].log_data[9].max := 1.0, [149].log_data[9].total := 523.749, [149].log_data[9].time := 3599.5, [149].log_data[9].maxminute := 51, [149].log_data[9].valid := 1, [149].log_data[10].min := 1.0, [149].log_data[10].max := 1.0, [149].log_data[10].total := 3599.5, [149].log_data[10].time := 3599.5, [149].log_data[10].valid := 1, [149].log_data[11].time := 3599.5, [149].log_data[11].valid := 1, [149].log_data[12].min := 1.0, [149].log_data[12].max := 1.0, [149].log_data[12].total := 3599.5, [149].log_data[12].time := 3599.5, [149].log_data[12].valid := 1, [149].log_data[13].min := 1.0, [149].log_data[13].max := 1.0, [149].log_data[13].total := 3599.5, [149].log_data[13].time := 3599.5, [149].log_data[13].valid := 1, [149].log_data[14].time := 3599.5, [149].log_data[14].valid := 1, [149].log_data[15].time := 3599.5, [149].log_data[15].valid := 1, [149].log_data[16].time := 3599.5, [149].log_data[16].valid := 1, [149].log_data[17].min := 1.0, [149].log_data[17].max := 1.0, [149].log_data[17].total := 3599.5, [149].log_data[17].time := 3599.5, [149].log_data[17].valid := 1, [149].log_data[18].time := 3599.5, [149].log_data[18].valid := 1, [149].log_data[19].time := 3599.5, [149].log_data[19].valid := 1, [149].log_data[20].time := 3599.5, [149].log_data[20].valid := 1, [149].log_data[21].min := 1.0, [149].log_data[21].max := 1.0, [149].log_data[21].total := 3599.5, [149].log_data[21].time := 3599.5, [149].log_data[21].valid := 1, [149].log_data[22].time := 3599.5, [149].log_data[22].valid := 1, [149].log_data[23].time := 3599.5, [149].log_data[23].valid := 1, [149].log_data[24].time := 3599.5, [149].log_data[24].valid := 1,
        [149].log_data[25].time := 3599.5, [149].log_data[25].valid := 1, [149].log_data[26].time := 3599.5, [149].log_data[26].valid := 1, [149].log_data[27].time := 3599.5, [149].log_data[27].valid := 1, [149].log_data[28].time := 3599.5, [149].log_data[28].valid := 1, [149].log_data[29].min := 1.0, [149].log_data[29].max := 1.0, [149].log_data[29].total := 3599.5, [149].log_data[29].time := 3599.5, [149].log_data[29].valid := 1, [149].log_data[30].min := 1.0, [149].log_data[30].max := 1.0, [149].log_data[30].total := 3599.5, [149].log_data[30].time := 3599.5, [149].log_data[30].valid := 1, [149].log_data[31].max := 1.0, [149].log_data[31].total := 520.249, [149].log_data[31].time := 3599.5, [149].log_data[31].maxminute := 51, [149].log_data[31].valid := 1, [149].log_data[32].time := 3599.5, [149].log_data[32].valid := 1, [149].log_data[33].time := 3599.5, [149].log_data[33].valid := 1, [149].log_data[34].time := 3599.5, [149].log_data[34].valid := 1, [149].log_data[35].max := 1.0, [149].log_data[35].total := 85.749, [149].log_data[35].time := 3599.5, [149].log_data[35].maxminute := 58, [149].log_data[35].valid := 1, [149].log_data[36].max := 1.0, [149].log_data[36].total := 342.749, [149].log_data[36].time := 3599.5, [149].log_data[36].maxminute := 51, [149].log_data[36].valid := 1, [149].log_data[37].max := 7.239552, [149].log_data[37].total := 3586.8643, [149].log_data[37].time := 3599.5, [149].log_data[37].maxminute := 48, [149].log_data[37].valid := 1, [149].log_data[38].time := 3599.5, [149].log_data[38].valid := 1, [149].log_data[39].min := 0.9947063, [149].log_data[39].max := 1.0226188, [149].log_data[39].total := 3608.074, [149].log_data[39].time := 3599.5, [149].log_data[39].minminute := 43, [149].log_data[39].maxminute := 54, [149].log_data[39].valid := 1, [149].log_data[40].min := 7.5942707, [149].log_data[40].max := 7.6275225, [149].log_data[40].total := 27400.95, [149].log_data[40].time := 3599.5, [149].log_data[40].minminute := 17, [149].log_data[40].maxminute := 56, [149].log_data[40].valid := 1,
        [149].log_data[41].min := 0.02273633, [149].log_data[41].max := 0.023128908, [149].log_data[41].total := 82.43481, [149].log_data[41].time := 3599.5, [149].log_data[41].valid := 1, [149].log_data[42].min := 2.291407, [149].log_data[42].max := 2.2960005, [149].log_data[42].total := 8256.407, [149].log_data[42].time := 3599.5, [149].log_data[42].minminute := 15, [149].log_data[42].maxminute := 39, [149].log_data[42].valid := 1, [149].log_data[43].min := -0.27999878, [149].log_data[43].max := -0.26000214, [149].log_data[43].total := -935.8482, [149].log_data[43].time := 3599.5, [149].log_data[43].minminute := 36, [149].log_data[43].valid := 1, [149].log_data[44].min := -0.30000305, [149].log_data[44].max := -0.27999878, [149].log_data[44].total := -1072.455, [149].log_data[44].time := 3599.5, [149].log_data[44].valid := 1, [149].log_data[45].time := 3599.5, [149].log_data[45].valid := 1, [149].log_data[46].time := 3599.5, [149].log_data[46].valid := 1, [149].log_data[47].time := 3599.5, [149].log_data[47].valid := 1, [149].log_data[48].min := 6.676412, [149].log_data[48].max := 6.916595, [149].log_data[48].total := 24159.102, [149].log_data[48].time := 3599.5, [149].log_data[48].maxminute := 57, [149].log_data[48].valid := 1, [149].log_data[49].min := 8.366299, [149].log_data[49].max := 9.761538, [149].log_data[49].total := 34677.277, [149].log_data[49].time := 3599.5, [149].log_data[49].minminute := 59, [149].log_data[49].maxminute := 50, [149].log_data[49].valid := 1, [149].log_data[50].min := 2.0653973, [149].log_data[50].max := 2.151373, [149].log_data[50].total := 7622.6294, [149].log_data[50].time := 3599.5, [149].log_data[50].minminute := 54, [149].log_data[50].maxminute := 51, [149].log_data[50].valid := 1, [149].log_data[51].time := 3599.5, [149].log_data[51].valid := 1, [149].log_data[52].min := -4.159996, [149].log_data[52].max := -1.4599991, [149].log_data[52].total := -6095.813, [149].log_data[52].time := 3599.5, [149].log_data[52].minminute := 51, [149].log_data[52].maxminute := 28, [149].log_data[52].valid := 1, [149].log_data[53].min := -3.9399948, [149].log_data[53].max := 0.44000244,
        [149].log_data[53].total := -5477.128, [149].log_data[53].time := 3599.5, [149].log_data[53].minminute := 51, [149].log_data[53].maxminute := 58, [149].log_data[53].valid := 1, [149].log_data[54].max := 0.508, [149].log_data[54].total := 205.80003, [149].log_data[54].time := 3599.5, [149].log_data[54].maxminute := 51, [149].log_data[54].valid := 1, [149].log_data[55].max := 0.506, [149].log_data[55].total := 167.42897, [149].log_data[55].time := 3599.5, [149].log_data[55].maxminute := 58, [149].log_data[55].valid := 1, [149].log_data[56].min := 0.15910713, [149].log_data[56].max := 0.15953897, [149].log_data[56].total := 573.3672, [149].log_data[56].time := 3599.5, [149].log_data[56].minminute := 25, [149].log_data[56].maxminute := 19, [149].log_data[56].valid := 1, [149].log_data[57].min := 0.19349736, [149].log_data[57].max := 0.19388995, [149].log_data[57].total := 696.9809, [149].log_data[57].time := 3599.5, [149].log_data[57].minminute := 25, [149].log_data[57].maxminute := 8, [149].log_data[57].valid := 1, [149].log_data[58].time := 3599.5, [149].log_data[58].valid := 1, [149].log_data[59].time := 3599.5, [149].log_data[59].valid := 1, [149].log_data[60].valid := 1, [149].log_data[61].valid := 1, [149].log_data[62].valid := 1, [149].log_data[63].valid := 1, [149].log_data[64].valid := 1, [149].log_data[65].valid := 1, [149].log_data[66].valid := 1, [149].log_data[67].valid := 1, [149].log_data[68].valid := 1, [149].log_data[69].valid := 1, [149].log_data[70].valid := 1, [149].log_data[71].valid := 1, [149].log_data[72].valid := 1, [149].log_data[73].valid := 1, [149].log_data[74].valid := 1, [149].log_data[75].valid := 1, [149].log_data[76].valid := 1, [149].log_data[77].valid := 1, [149].log_data[78].valid := 1, [149].log_data[79].valid := 1, [149].log_data[80].valid := 1, [149].log_data[81].valid := 1, [149].log_data[82].valid := 1, [149].log_data[83].valid := 1, [149].log_data[84].valid := 1, [149].log_data[85].valid := 1, [149].log_data[86].valid := 1,
        [149].log_data[87].valid := 1, [149].log_data[88].valid := 1, [149].log_data[89].valid := 1, [149].log_data[90].valid := 1, [149].log_data[91].valid := 1, [149].log_data[92].valid := 1, [149].log_data[93].valid := 1, [149].log_data[94].valid := 1, [149].log_data[95].valid := 1, [149].log_data[96].valid := 1, [149].log_data[97].valid := 1, [149].log_data[98].valid := 1, [149].log_data[99].valid := 1, [149].log_data[100].valid := 1, [149].log_data[101].valid := 1, [149].log_data[102].valid := 1, [149].log_data[103].valid := 1, [149].log_data[104].valid := 1, [149].log_data[105].valid := 1, [149].log_data[106].valid := 1, [149].log_data[107].valid := 1, [149].log_data[108].valid := 1, [149].log_data[109].valid := 1, [149].log_data[110].valid := 1, [149].log_data[111].valid := 1, [149].log_data[112].valid := 1, [149].log_data[113].valid := 1, [149].log_data[114].valid := 1, [149].log_data[115].valid := 1, [149].log_data[116].valid := 1, [149].log_data[117].valid := 1, [149].log_data[118].valid := 1, [149].log_data[119].valid := 1, [149].log_data[120].valid := 1, [149].log_data[121].valid := 1, [149].log_data[122].valid := 1, [149].log_data[123].valid := 1, [149].log_data[124].valid := 1, [149].time.Year := 2023, [149].time.Month := 1, [149].time.Day := 19, [149].time.Hour := 8, [149].time.Minute := 59, [149].time.Second := 59, [150].log_data[0].min := 1.0, [150].log_data[0].max := 1.0, [150].log_data[0].total := 3600.0, [150].log_data[0].time := 3600.0, [150].log_data[0].valid := 1, [150].log_data[1].max := 1.0, [150].log_data[1].total := 78.249, [150].log_data[1].time := 3600.0, [150].log_data[1].maxminute := 58, [150].log_data[1].valid := 1, [150].log_data[2].max := 1.0, [150].log_data[2].total := 74.749, [150].log_data[2].time := 3600.0, [150].log_data[2].maxminute := 58, [150].log_data[2].valid := 1, [150].log_data[3].time := 3600.0,
        [150].log_data[3].valid := 1, [150].log_data[4].time := 3600.0, [150].log_data[4].valid := 1, [150].log_data[5].time := 3600.0, [150].log_data[5].valid := 1, [150].log_data[6].time := 3600.0, [150].log_data[6].valid := 1, [150].log_data[7].time := 3600.0, [150].log_data[7].valid := 1, [150].log_data[8].min := 1.0, [150].log_data[8].max := 1.0, [150].log_data[8].total := 3600.0, [150].log_data[8].time := 3600.0, [150].log_data[8].valid := 1, [150].log_data[9].min := 1.0, [150].log_data[9].max := 1.0, [150].log_data[9].total := 3600.0, [150].log_data[9].time := 3600.0, [150].log_data[9].valid := 1, [150].log_data[10].min := 1.0, [150].log_data[10].max := 1.0, [150].log_data[10].total := 3600.0, [150].log_data[10].time := 3600.0, [150].log_data[10].valid := 1, [150].log_data[11].time := 3600.0, [150].log_data[11].valid := 1, [150].log_data[12].min := 1.0, [150].log_data[12].max := 1.0, [150].log_data[12].total := 3600.0, [150].log_data[12].time := 3600.0, [150].log_data[12].valid := 1, [150].log_data[13].min := 1.0, [150].log_data[13].max := 1.0, [150].log_data[13].total := 3600.0, [150].log_data[13].time := 3600.0, [150].log_data[13].valid := 1, [150].log_data[14].time := 3600.0, [150].log_data[14].valid := 1, [150].log_data[15].time := 3600.0, [150].log_data[15].valid := 1, [150].log_data[16].time := 3600.0, [150].log_data[16].valid := 1, [150].log_data[17].min := 1.0, [150].log_data[17].max := 1.0, [150].log_data[17].total := 3600.0, [150].log_data[17].time := 3600.0, [150].log_data[17].valid := 1, [150].log_data[18].time := 3600.0, [150].log_data[18].valid := 1, [150].log_data[19].time := 3600.0, [150].log_data[19].valid := 1, [150].log_data[20].time := 3600.0, [150].log_data[20].valid := 1, [150].log_data[21].min := 1.0, [150].log_data[21].max := 1.0, [150].log_data[21].total := 3600.0, [150].log_data[21].time := 3600.0, [150].log_data[21].valid := 1, [150].log_data[22].time := 3600.0, [150].log_data[22].valid := 1,
        [150].log_data[23].time := 3600.0, [150].log_data[23].valid := 1, [150].log_data[24].time := 3600.0, [150].log_data[24].valid := 1, [150].log_data[25].time := 3600.0, [150].log_data[25].valid := 1, [150].log_data[26].time := 3600.0, [150].log_data[26].valid := 1, [150].log_data[27].time := 3600.0, [150].log_data[27].valid := 1, [150].log_data[28].time := 3600.0, [150].log_data[28].valid := 1, [150].log_data[29].min := 1.0, [150].log_data[29].max := 1.0, [150].log_data[29].total := 3600.0, [150].log_data[29].time := 3600.0, [150].log_data[29].valid := 1, [150].log_data[30].min := 1.0, [150].log_data[30].max := 1.0, [150].log_data[30].total := 3600.0, [150].log_data[30].time := 3600.0, [150].log_data[30].valid := 1, [150].log_data[31].max := 1.0, [150].log_data[31].total := 1440.498, [150].log_data[31].time := 3600.0, [150].log_data[31].valid := 1, [150].log_data[32].max := 1.0, [150].log_data[32].total := 1630.249, [150].log_data[32].time := 3600.0, [150].log_data[32].maxminute := 1, [150].log_data[32].valid := 1, [150].log_data[33].time := 3600.0, [150].log_data[33].valid := 1, [150].log_data[34].time := 3600.0, [150].log_data[34].valid := 1, [150].log_data[35].max := 1.0, [150].log_data[35].total := 1543.998, [150].log_data[35].time := 3600.0, [150].log_data[35].minminute := 7, [150].log_data[35].valid := 1, [150].log_data[36].max := 1.0, [150].log_data[36].total := 1614.7471, [150].log_data[36].time := 3600.0, [150].log_data[36].maxminute := 9, [150].log_data[36].valid := 1, [150].log_data[37].max := 7.521034, [150].log_data[37].total := 570.2758, [150].log_data[37].time := 3600.0, [150].log_data[37].maxminute := 59, [150].log_data[37].valid := 1, [150].log_data[38].time := 3600.0, [150].log_data[38].valid := 1, [150].log_data[39].min := 0.9936463, [150].log_data[39].max := 1.0087214, [150].log_data[39].total := 3598.4565, [150].log_data[39].time := 3600.0, [150].log_data[39].minminute := 48, [150].log_data[39].maxminute := 59, [150].log_data[39].valid := 1, [150].log_data[40].min := 7.579981,
        [150].log_data[40].max := 7.6244993, [150].log_data[40].total := 27411.877, [150].log_data[40].time := 3600.0, [150].log_data[40].minminute := 7, [150].log_data[40].maxminute := 11, [150].log_data[40].valid := 1, [150].log_data[41].min := 0.022540038, [150].log_data[41].max := 0.023128908, [150].log_data[41].total := 82.42599, [150].log_data[41].time := 3600.0, [150].log_data[41].minminute := 52, [150].log_data[41].valid := 1, [150].log_data[42].min := 2.2910538, [150].log_data[42].max := 2.296118, [150].log_data[42].total := 8257.579, [150].log_data[42].time := 3600.0, [150].log_data[42].minminute := 11, [150].log_data[42].maxminute := 45, [150].log_data[42].valid := 1, [150].log_data[43].min := -0.26000214, [150].log_data[43].max := -0.26000214, [150].log_data[43].total := -935.9732, [150].log_data[43].time := 3600.0, [150].log_data[43].valid := 1, [150].log_data[44].min := -0.30000305, [150].log_data[44].max := -0.27999878, [150].log_data[44].total := -1064.3453, [150].log_data[44].time := 3600.0, [150].log_data[44].valid := 1, [150].log_data[45].time := 3600.0, [150].log_data[45].valid := 1, [150].log_data[46].time := 3600.0, [150].log_data[46].valid := 1, [150].log_data[47].time := 3600.0, [150].log_data[47].valid := 1, [150].log_data[48].min := 6.5678625, [150].log_data[48].max := 6.815465, [150].log_data[48].total := 24173.568, [150].log_data[48].time := 3600.0, [150].log_data[48].minminute := 16, [150].log_data[48].maxminute := 32, [150].log_data[48].valid := 1, [150].log_data[49].min := 6.997362, [150].log_data[49].max := 9.520294, [150].log_data[49].total := 29569.84, [150].log_data[49].time := 3600.0, [150].log_data[49].minminute := 15, [150].log_data[49].maxminute := 58, [150].log_data[49].valid := 1, [150].log_data[50].min := 2.037249, [150].log_data[50].max := 2.1234603, [150].log_data[50].total := 7497.493, [150].log_data[50].time := 3600.0, [150].log_data[50].minminute := 59, [150].log_data[50].maxminute := 2, [150].log_data[50].valid := 1, [150].log_data[51].time := 3600.0, [150].log_data[51].valid := 1, [150].log_data[52].min := -2.8600006, [150].log_data[52].max := 0.11999512,
        [150].log_data[52].total := -7488.6313, [150].log_data[52].time := 3600.0, [150].log_data[52].minminute := 22, [150].log_data[52].valid := 1, [150].log_data[53].min := -2.4200058, [150].log_data[53].max := 0.3600006, [150].log_data[53].total := -6774.6255, [150].log_data[53].time := 3600.0, [150].log_data[53].minminute := 27, [150].log_data[53].maxminute := 8, [150].log_data[53].valid := 1, [150].log_data[54].max := 0.5565, [150].log_data[54].total := 1217.2712, [150].log_data[54].time := 3600.0, [150].log_data[54].maxminute := 54, [150].log_data[54].valid := 1, [150].log_data[55].max := 0.502, [150].log_data[55].total := 1254.1625, [150].log_data[55].time := 3600.0, [150].log_data[55].minminute := 7, [150].log_data[55].maxminute := 30, [150].log_data[55].valid := 1, [150].log_data[56].min := 0.15902862, [150].log_data[56].max := 0.1594997, [150].log_data[56].total := 573.2354, [150].log_data[56].time := 3600.0, [150].log_data[56].minminute := 15, [150].log_data[56].maxminute := 1, [150].log_data[56].valid := 1, [150].log_data[57].min := 0.19149521, [150].log_data[57].max := 0.19385068, [150].log_data[57].total := 692.236, [150].log_data[57].time := 3600.0, [150].log_data[57].minminute := 29, [150].log_data[57].maxminute := 1, [150].log_data[57].valid := 1, [150].log_data[58].time := 3600.0, [150].log_data[58].valid := 1, [150].log_data[59].time := 3600.0, [150].log_data[59].valid := 1, [150].log_data[60].valid := 1, [150].log_data[61].valid := 1, [150].log_data[62].valid := 1, [150].log_data[63].valid := 1, [150].log_data[64].valid := 1, [150].log_data[65].valid := 1, [150].log_data[66].valid := 1, [150].log_data[67].valid := 1, [150].log_data[68].valid := 1, [150].log_data[69].valid := 1, [150].log_data[70].valid := 1, [150].log_data[71].valid := 1, [150].log_data[72].valid := 1, [150].log_data[73].valid := 1, [150].log_data[74].valid := 1, [150].log_data[75].valid := 1, [150].log_data[76].valid := 1, [150].log_data[77].valid := 1, [150].log_data[78].valid := 1, [150].log_data[79].valid := 1,
        [150].log_data[80].valid := 1, [150].log_data[81].valid := 1, [150].log_data[82].valid := 1, [150].log_data[83].valid := 1, [150].log_data[84].valid := 1, [150].log_data[85].valid := 1, [150].log_data[86].valid := 1, [150].log_data[87].valid := 1, [150].log_data[88].valid := 1, [150].log_data[89].valid := 1, [150].log_data[90].valid := 1, [150].log_data[91].valid := 1, [150].log_data[92].valid := 1, [150].log_data[93].valid := 1, [150].log_data[94].valid := 1, [150].log_data[95].valid := 1, [150].log_data[96].valid := 1, [150].log_data[97].valid := 1, [150].log_data[98].valid := 1, [150].log_data[99].valid := 1, [150].log_data[100].valid := 1, [150].log_data[101].valid := 1, [150].log_data[102].valid := 1, [150].log_data[103].valid := 1, [150].log_data[104].valid := 1, [150].log_data[105].valid := 1, [150].log_data[106].valid := 1, [150].log_data[107].valid := 1, [150].log_data[108].valid := 1, [150].log_data[109].valid := 1, [150].log_data[110].valid := 1, [150].log_data[111].valid := 1, [150].log_data[112].valid := 1, [150].log_data[113].valid := 1, [150].log_data[114].valid := 1, [150].log_data[115].valid := 1, [150].log_data[116].valid := 1, [150].log_data[117].valid := 1, [150].log_data[118].valid := 1, [150].log_data[119].valid := 1, [150].log_data[120].valid := 1, [150].log_data[121].valid := 1, [150].log_data[122].valid := 1, [150].log_data[123].valid := 1, [150].log_data[124].valid := 1, [150].time.Year := 2023, [150].time.Month := 1, [150].time.Day := 19, [150].time.Hour := 9, [150].time.Minute := 59, [150].time.Second := 59, [151].log_data[0].min := 1.0, [151].log_data[0].max := 1.0, [151].log_data[0].total := 3600.0, [151].log_data[0].time := 3600.0, [151].log_data[0].valid := 1, [151].log_data[1].max := 1.0, [151].log_data[1].total := 462.751, [151].log_data[1].time := 3600.0, [151].log_data[1].minminute := 7,
        [151].log_data[1].valid := 1, [151].log_data[2].max := 1.0, [151].log_data[2].total := 462.751, [151].log_data[2].time := 3600.0, [151].log_data[2].minminute := 7, [151].log_data[2].valid := 1, [151].log_data[3].time := 3600.0, [151].log_data[3].valid := 1, [151].log_data[4].time := 3600.0, [151].log_data[4].valid := 1, [151].log_data[5].max := 1.0, [151].log_data[5].total := 233.5, [151].log_data[5].time := 3600.0, [151].log_data[5].maxminute := 1, [151].log_data[5].valid := 1, [151].log_data[6].time := 3600.0, [151].log_data[6].valid := 1, [151].log_data[7].time := 3600.0, [151].log_data[7].valid := 1, [151].log_data[8].min := 1.0, [151].log_data[8].max := 1.0, [151].log_data[8].total := 3600.0, [151].log_data[8].time := 3600.0, [151].log_data[8].valid := 1, [151].log_data[9].min := 1.0, [151].log_data[9].max := 1.0, [151].log_data[9].total := 3600.0, [151].log_data[9].time := 3600.0, [151].log_data[9].valid := 1, [151].log_data[10].min := 1.0, [151].log_data[10].max := 1.0, [151].log_data[10].total := 3600.0, [151].log_data[10].time := 3600.0, [151].log_data[10].valid := 1, [151].log_data[11].time := 3600.0, [151].log_data[11].valid := 1, [151].log_data[12].min := 1.0, [151].log_data[12].max := 1.0, [151].log_data[12].total := 3600.0, [151].log_data[12].time := 3600.0, [151].log_data[12].valid := 1, [151].log_data[13].min := 1.0, [151].log_data[13].max := 1.0, [151].log_data[13].total := 3600.0, [151].log_data[13].time := 3600.0, [151].log_data[13].valid := 1, [151].log_data[14].time := 3600.0, [151].log_data[14].valid := 1, [151].log_data[15].time := 3600.0, [151].log_data[15].valid := 1, [151].log_data[16].time := 3600.0, [151].log_data[16].valid := 1, [151].log_data[17].min := 1.0, [151].log_data[17].max := 1.0, [151].log_data[17].total := 3600.0, [151].log_data[17].time := 3600.0, [151].log_data[17].valid := 1, [151].log_data[18].time := 3600.0, [151].log_data[18].valid := 1, [151].log_data[19].time := 3600.0,
        [151].log_data[19].valid := 1, [151].log_data[20].time := 3600.0, [151].log_data[20].valid := 1, [151].log_data[21].min := 1.0, [151].log_data[21].max := 1.0, [151].log_data[21].total := 3600.0, [151].log_data[21].time := 3600.0, [151].log_data[21].valid := 1, [151].log_data[22].time := 3600.0, [151].log_data[22].valid := 1, [151].log_data[23].time := 3600.0, [151].log_data[23].valid := 1, [151].log_data[24].time := 3600.0, [151].log_data[24].valid := 1, [151].log_data[25].time := 3600.0, [151].log_data[25].valid := 1, [151].log_data[26].time := 3600.0, [151].log_data[26].valid := 1, [151].log_data[27].time := 3600.0, [151].log_data[27].valid := 1, [151].log_data[28].time := 3600.0, [151].log_data[28].valid := 1, [151].log_data[29].min := 1.0, [151].log_data[29].max := 1.0, [151].log_data[29].total := 3600.0, [151].log_data[29].time := 3600.0, [151].log_data[29].valid := 1, [151].log_data[30].min := 1.0, [151].log_data[30].max := 1.0, [151].log_data[30].total := 3600.0, [151].log_data[30].time := 3600.0, [151].log_data[30].valid := 1, [151].log_data[31].max := 1.0, [151].log_data[31].total := 1440.7471, [151].log_data[31].time := 3600.0, [151].log_data[31].minminute := 3, [151].log_data[31].valid := 1, [151].log_data[32].max := 1.0, [151].log_data[32].total := 1629.998, [151].log_data[32].time := 3600.0, [151].log_data[32].maxminute := 5, [151].log_data[32].valid := 1, [151].log_data[33].time := 3600.0, [151].log_data[33].valid := 1, [151].log_data[34].time := 3600.0, [151].log_data[34].valid := 1, [151].log_data[35].max := 1.0, [151].log_data[35].total := 1629.998, [151].log_data[35].time := 3600.0, [151].log_data[35].maxminute := 1, [151].log_data[35].valid := 1, [151].log_data[36].max := 1.0, [151].log_data[36].total := 1440.2471, [151].log_data[36].time := 3600.0, [151].log_data[36].valid := 1, [151].log_data[37].max := 7.560685, [151].log_data[37].total := 2984.308, [151].log_data[37].time := 3600.0, [151].log_data[37].minminute := 6, [151].log_data[37].maxminute := 1,
        [151].log_data[37].valid := 1, [151].log_data[38].time := 3600.0, [151].log_data[38].valid := 1, [151].log_data[39].min := 0.995884, [151].log_data[39].max := 1.0207345, [151].log_data[39].total := 3606.8933, [151].log_data[39].time := 3600.0, [151].log_data[39].minminute := 58, [151].log_data[39].maxminute := 1, [151].log_data[39].valid := 1, [151].log_data[40].min := 7.608561, [151].log_data[40].max := 7.621752, [151].log_data[40].total := 27416.006, [151].log_data[40].time := 3600.0, [151].log_data[40].minminute := 52, [151].log_data[40].maxminute := 3, [151].log_data[40].valid := 1, [151].log_data[41].min := 0.022540038, [151].log_data[41].max := 0.023128908, [151].log_data[41].total := 82.45791, [151].log_data[41].time := 3600.0, [151].log_data[41].minminute := 53, [151].log_data[41].valid := 1, [151].log_data[42].min := 2.2910538, [151].log_data[42].max := 2.2960005, [151].log_data[42].total := 8257.643, [151].log_data[42].time := 3600.0, [151].log_data[42].minminute := 43, [151].log_data[42].maxminute := 22, [151].log_data[42].valid := 1, [151].log_data[43].min := -0.27999878, [151].log_data[43].max := -0.26000214, [151].log_data[43].total := -935.9782, [151].log_data[43].time := 3600.0, [151].log_data[43].minminute := 16, [151].log_data[43].valid := 1, [151].log_data[44].min := -0.30000305, [151].log_data[44].max := -0.27999878, [151].log_data[44].total := -1069.9171, [151].log_data[44].time := 3600.0, [151].log_data[44].valid := 1, [151].log_data[45].time := 3600.0, [151].log_data[45].valid := 1, [151].log_data[46].time := 3600.0, [151].log_data[46].valid := 1, [151].log_data[47].time := 3600.0, [151].log_data[47].valid := 1, [151].log_data[48].min := 6.5722604, [151].log_data[48].max := 6.936381, [151].log_data[48].total := 24216.379, [151].log_data[48].time := 3600.0, [151].log_data[48].minminute := 29, [151].log_data[48].maxminute := 4, [151].log_data[48].valid := 1, [151].log_data[49].min := 6.9412227, [151].log_data[49].max := 9.54699, [151].log_data[49].total := 29156.982, [151].log_data[49].time := 3600.0, [151].log_data[49].minminute := 29, [151].log_data[49].maxminute := 1,
        [151].log_data[49].valid := 1, [151].log_data[50].min := 2.0370135, [151].log_data[50].max := 2.1458375, [151].log_data[50].total := 7588.35, [151].log_data[50].time := 3600.0, [151].log_data[50].maxminute := 8, [151].log_data[50].valid := 1, [151].log_data[51].time := 3600.0, [151].log_data[51].valid := 1, [151].log_data[52].min := -2.7400055, [151].log_data[52].max := 0.11999512, [151].log_data[52].total := -7495.446, [151].log_data[52].time := 3600.0, [151].log_data[52].minminute := 36, [151].log_data[52].maxminute := 3, [151].log_data[52].valid := 1, [151].log_data[53].min := -2.540001, [151].log_data[53].max := 0.38000488, [151].log_data[53].total := -6610.2627, [151].log_data[53].time := 3600.0, [151].log_data[53].minminute := 54, [151].log_data[53].maxminute := 33, [151].log_data[53].valid := 1, [151].log_data[54].max := 0.544, [151].log_data[54].total := 1217.0946, [151].log_data[54].time := 3600.0, [151].log_data[54].minminute := 3, [151].log_data[54].maxminute := 36, [151].log_data[54].valid := 1, [151].log_data[55].max := 0.5545, [151].log_data[55].total := 1217.5413, [151].log_data[55].time := 3600.0, [151].log_data[55].maxminute := 54, [151].log_data[55].valid := 1, [151].log_data[56].min := 0.15895009, [151].log_data[56].max := 0.1594997, [151].log_data[56].total := 573.1523, [151].log_data[56].time := 3600.0, [151].log_data[56].minminute := 4, [151].log_data[56].maxminute := 6, [151].log_data[56].valid := 1, [151].log_data[57].min := 0.18953228, [151].log_data[57].max := 0.1918878, [151].log_data[57].total := 686.5759, [151].log_data[57].time := 3600.0, [151].log_data[57].minminute := 52, [151].log_data[57].maxminute := 3, [151].log_data[57].valid := 1, [151].log_data[58].time := 3600.0, [151].log_data[58].valid := 1, [151].log_data[59].time := 3600.0, [151].log_data[59].valid := 1, [151].log_data[60].valid := 1, [151].log_data[61].valid := 1, [151].log_data[62].valid := 1, [151].log_data[63].valid := 1, [151].log_data[64].valid := 1, [151].log_data[65].valid := 1, [151].log_data[66].valid := 1, [151].log_data[67].valid := 1,
        [151].log_data[68].valid := 1, [151].log_data[69].valid := 1, [151].log_data[70].valid := 1, [151].log_data[71].valid := 1, [151].log_data[72].valid := 1, [151].log_data[73].valid := 1, [151].log_data[74].valid := 1, [151].log_data[75].valid := 1, [151].log_data[76].valid := 1, [151].log_data[77].valid := 1, [151].log_data[78].valid := 1, [151].log_data[79].valid := 1, [151].log_data[80].valid := 1, [151].log_data[81].valid := 1, [151].log_data[82].valid := 1, [151].log_data[83].valid := 1, [151].log_data[84].valid := 1, [151].log_data[85].valid := 1, [151].log_data[86].valid := 1, [151].log_data[87].valid := 1, [151].log_data[88].valid := 1, [151].log_data[89].valid := 1, [151].log_data[90].valid := 1, [151].log_data[91].valid := 1, [151].log_data[92].valid := 1, [151].log_data[93].valid := 1, [151].log_data[94].valid := 1, [151].log_data[95].valid := 1, [151].log_data[96].valid := 1, [151].log_data[97].valid := 1, [151].log_data[98].valid := 1, [151].log_data[99].valid := 1, [151].log_data[100].valid := 1, [151].log_data[101].valid := 1, [151].log_data[102].valid := 1, [151].log_data[103].valid := 1, [151].log_data[104].valid := 1, [151].log_data[105].valid := 1, [151].log_data[106].valid := 1, [151].log_data[107].valid := 1, [151].log_data[108].valid := 1, [151].log_data[109].valid := 1, [151].log_data[110].valid := 1, [151].log_data[111].valid := 1, [151].log_data[112].valid := 1, [151].log_data[113].valid := 1, [151].log_data[114].valid := 1, [151].log_data[115].valid := 1, [151].log_data[116].valid := 1, [151].log_data[117].valid := 1, [151].log_data[118].valid := 1, [151].log_data[119].valid := 1, [151].log_data[120].valid := 1, [151].log_data[121].valid := 1, [151].log_data[122].valid := 1, [151].log_data[123].valid := 1, [151].log_data[124].valid := 1, [151].time.Year := 2023, [151].time.Month := 1, [151].time.Day := 19,
        [151].time.Hour := 10, [151].time.Minute := 59, [151].time.Second := 59, [152].log_data[0].min := 1.0, [152].log_data[0].max := 1.0, [152].log_data[0].total := 3600.0, [152].log_data[0].time := 3600.0, [152].log_data[0].valid := 1, [152].log_data[1].max := 1.0, [152].log_data[1].total := 566.5, [152].log_data[1].time := 3600.0, [152].log_data[1].maxminute := 43, [152].log_data[1].valid := 1, [152].log_data[2].max := 1.0, [152].log_data[2].total := 563.0, [152].log_data[2].time := 3600.0, [152].log_data[2].maxminute := 43, [152].log_data[2].valid := 1, [152].log_data[3].time := 3600.0, [152].log_data[3].valid := 1, [152].log_data[4].time := 3600.0, [152].log_data[4].valid := 1, [152].log_data[5].max := 1.0, [152].log_data[5].total := 239.0, [152].log_data[5].time := 3600.0, [152].log_data[5].maxminute := 46, [152].log_data[5].valid := 1, [152].log_data[6].time := 3600.0, [152].log_data[6].valid := 1, [152].log_data[7].time := 3600.0, [152].log_data[7].valid := 1, [152].log_data[8].min := 1.0, [152].log_data[8].max := 1.0, [152].log_data[8].total := 3600.0, [152].log_data[8].time := 3600.0, [152].log_data[8].valid := 1, [152].log_data[9].min := 1.0, [152].log_data[9].max := 1.0, [152].log_data[9].total := 3600.0, [152].log_data[9].time := 3600.0, [152].log_data[9].valid := 1, [152].log_data[10].min := 1.0, [152].log_data[10].max := 1.0, [152].log_data[10].total := 3600.0, [152].log_data[10].time := 3600.0, [152].log_data[10].valid := 1, [152].log_data[11].time := 3600.0, [152].log_data[11].valid := 1, [152].log_data[12].min := 1.0, [152].log_data[12].max := 1.0, [152].log_data[12].total := 3600.0, [152].log_data[12].time := 3600.0, [152].log_data[12].valid := 1, [152].log_data[13].min := 1.0, [152].log_data[13].max := 1.0, [152].log_data[13].total := 3600.0, [152].log_data[13].time := 3600.0, [152].log_data[13].valid := 1, [152].log_data[14].time := 3600.0, [152].log_data[14].valid := 1,
        [152].log_data[15].time := 3600.0, [152].log_data[15].valid := 1, [152].log_data[16].time := 3600.0, [152].log_data[16].valid := 1, [152].log_data[17].min := 1.0, [152].log_data[17].max := 1.0, [152].log_data[17].total := 3600.0, [152].log_data[17].time := 3600.0, [152].log_data[17].valid := 1, [152].log_data[18].time := 3600.0, [152].log_data[18].valid := 1, [152].log_data[19].time := 3600.0, [152].log_data[19].valid := 1, [152].log_data[20].time := 3600.0, [152].log_data[20].valid := 1, [152].log_data[21].min := 1.0, [152].log_data[21].max := 1.0, [152].log_data[21].total := 3600.0, [152].log_data[21].time := 3600.0, [152].log_data[21].valid := 1, [152].log_data[22].time := 3600.0, [152].log_data[22].valid := 1, [152].log_data[23].time := 3600.0, [152].log_data[23].valid := 1, [152].log_data[24].time := 3600.0, [152].log_data[24].valid := 1, [152].log_data[25].time := 3600.0, [152].log_data[25].valid := 1, [152].log_data[26].time := 3600.0, [152].log_data[26].valid := 1, [152].log_data[27].time := 3600.0, [152].log_data[27].valid := 1, [152].log_data[28].time := 3600.0, [152].log_data[28].valid := 1, [152].log_data[29].min := 1.0, [152].log_data[29].max := 1.0, [152].log_data[29].total := 3600.0, [152].log_data[29].time := 3600.0, [152].log_data[29].valid := 1, [152].log_data[30].max := 1.0, [152].log_data[30].total := 3542.0, [152].log_data[30].time := 3600.0, [152].log_data[30].minminute := 13, [152].log_data[30].valid := 1, [152].log_data[31].max := 1.0, [152].log_data[31].total := 1487.998, [152].log_data[31].time := 3600.0, [152].log_data[31].minminute := 6, [152].log_data[31].valid := 1, [152].log_data[32].max := 1.0, [152].log_data[32].total := 1629.7471, [152].log_data[32].time := 3600.0, [152].log_data[32].maxminute := 8, [152].log_data[32].valid := 1, [152].log_data[33].time := 3600.0, [152].log_data[33].valid := 1, [152].log_data[34].time := 3600.0, [152].log_data[34].valid := 1, [152].log_data[35].max := 1.0, [152].log_data[35].total := 1629.7471,
        [152].log_data[35].time := 3600.0, [152].log_data[35].maxminute := 4, [152].log_data[35].valid := 1, [152].log_data[36].max := 1.0, [152].log_data[36].total := 1440.7471, [152].log_data[36].time := 3600.0, [152].log_data[36].minminute := 3, [152].log_data[36].valid := 1, [152].log_data[37].max := 7.232486, [152].log_data[37].total := 3545.7905, [152].log_data[37].time := 3600.0, [152].log_data[37].maxminute := 44, [152].log_data[37].valid := 1, [152].log_data[38].time := 3600.0, [152].log_data[38].valid := 1, [152].log_data[39].min := 0.99494183, [152].log_data[39].max := 1.02097, [152].log_data[39].total := 3606.9504, [152].log_data[39].time := 3600.0, [152].log_data[39].maxminute := 51, [152].log_data[39].valid := 1, [152].log_data[40].min := 7.606912, [152].log_data[40].max := 7.621752, [152].log_data[40].total := 27413.89, [152].log_data[40].time := 3600.0, [152].log_data[40].minminute := 22, [152].log_data[40].maxminute := 24, [152].log_data[40].valid := 1, [152].log_data[41].min := 0.022343751, [152].log_data[41].max := 0.022932617, [152].log_data[41].total := 81.660866, [152].log_data[41].time := 3600.0, [152].log_data[41].minminute := 41, [152].log_data[41].valid := 1, [152].log_data[42].min := 2.290936, [152].log_data[42].max := 2.2964714, [152].log_data[42].total := 8257.459, [152].log_data[42].time := 3600.0, [152].log_data[42].minminute := 43, [152].log_data[42].maxminute := 35, [152].log_data[42].valid := 1, [152].log_data[43].min := -0.27999878, [152].log_data[43].max := -0.26000214, [152].log_data[43].total := -955.9954, [152].log_data[43].time := 3600.0, [152].log_data[43].minminute := 1, [152].log_data[43].valid := 1, [152].log_data[44].min := -0.30000305, [152].log_data[44].max := -0.27999878, [152].log_data[44].total := -1080.086, [152].log_data[44].time := 3600.0, [152].log_data[44].valid := 1, [152].log_data[45].time := 3600.0, [152].log_data[45].valid := 1, [152].log_data[46].time := 3600.0, [152].log_data[46].valid := 1, [152].log_data[47].time := 3600.0, [152].log_data[47].valid := 1, [152].log_data[48].min := 6.7102137, [152].log_data[48].max := 6.942976,
        [152].log_data[48].total := 24337.787, [152].log_data[48].time := 3600.0, [152].log_data[48].minminute := 59, [152].log_data[48].maxminute := 53, [152].log_data[48].valid := 1, [152].log_data[49].min := 7.549922, [152].log_data[49].max := 9.597437, [152].log_data[49].total := 33517.973, [152].log_data[49].time := 3600.0, [152].log_data[49].minminute := 59, [152].log_data[49].maxminute := 26, [152].log_data[49].valid := 1, [152].log_data[50].min := 2.0096898, [152].log_data[50].max := 2.1192203, [152].log_data[50].total := 7399.8315, [152].log_data[50].time := 3600.0, [152].log_data[50].minminute := 46, [152].log_data[50].maxminute := 54, [152].log_data[50].valid := 1, [152].log_data[51].time := 3600.0, [152].log_data[51].valid := 1, [152].log_data[52].min := -2.7400055, [152].log_data[52].max := 0.11999512, [152].log_data[52].total := -7653.7686, [152].log_data[52].time := 3600.0, [152].log_data[52].minminute := 8, [152].log_data[52].maxminute := 6, [152].log_data[52].valid := 1, [152].log_data[53].min := -2.5200043, [152].log_data[53].max := 0.32000732, [152].log_data[53].total := -6824.116, [152].log_data[53].time := 3600.0, [152].log_data[53].minminute := 4, [152].log_data[53].maxminute := 4, [152].log_data[53].valid := 1, [152].log_data[54].max := 0.5155, [152].log_data[54].total := 1238.4989, [152].log_data[54].time := 3600.0, [152].log_data[54].minminute := 6, [152].log_data[54].maxminute := 18, [152].log_data[54].valid := 1, [152].log_data[55].max := 0.557, [152].log_data[55].total := 1217.241, [152].log_data[55].time := 3600.0, [152].log_data[55].minminute := 3, [152].log_data[55].maxminute := 4, [152].log_data[55].valid := 1, [152].log_data[56].min := 0.15891084, [152].log_data[56].max := 0.15938194, [152].log_data[56].total := 572.8968, [152].log_data[56].time := 3600.0, [152].log_data[56].minminute := 42, [152].log_data[56].maxminute := 1, [152].log_data[56].valid := 1, [152].log_data[57].min := 0.18937525, [152].log_data[57].max := 0.18992485, [152].log_data[57].total := 682.66626, [152].log_data[57].time := 3600.0, [152].log_data[57].minminute := 57, [152].log_data[57].valid := 1,
